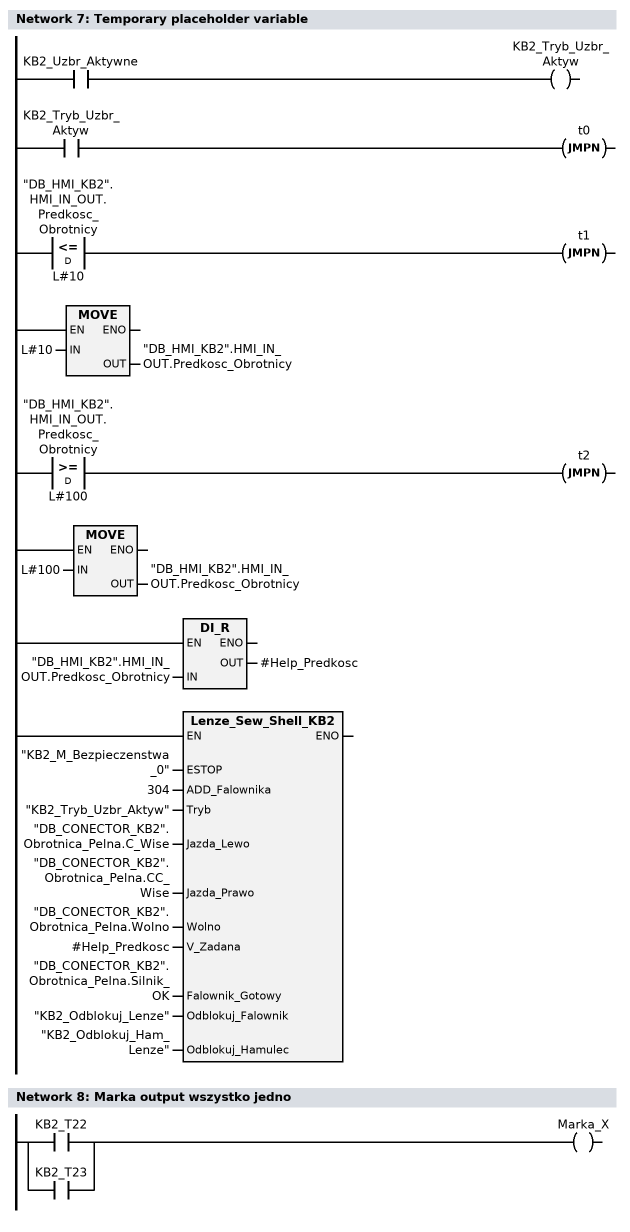
[picture p273: Przypis_Wyjsc_KB2 networks 7-8]
NETWORK
TITLE = Temporary placeholder variable
//Obrotnica Adres  9(Wirtualny)
// Dopasownie predkosci niskiej i wysokiej
      A     "KB2_Uzbr_Aktywne";
      =     "KB2_Tryb_Uzbr_Aktyw";
//************Przypisanie predkosci z panela*************
      A     "KB2_Tryb_Uzbr_Aktyw";
      JCN   t0;
//***Sprawdzenie czy predkosc nie jest za mala
      L     "DB_HMI_KB2".HMI_IN_OUT.Predkosc_Obrotnicy;
      L     L#10;
      <=D;
      JCN   t1;
      L     L#10;
      T     "DB_HMI_KB2".HMI_IN_OUT.Predkosc_Obrotnicy;
t1:   NOP   0;
//***Sprawdzenie czy predkosc nie jest za duza
      L     "DB_HMI_KB2".HMI_IN_OUT.Predkosc_Obrotnicy;
      L     L#100;
      >=D;
      JCN   t2;
      L     L#100;
      T     "DB_HMI_KB2".HMI_IN_OUT.Predkosc_Obrotnicy;
t2:   NOP   0;
//****Zamiana na real
t0:   NOP   0;
      L     "DB_HMI_KB2".HMI_IN_OUT.Predkosc_Obrotnicy;
      DTR;
      T     #Help_Predkosc;
//***Obsluga obrotnicy
      CALL  "Lenze_Sew_Shell_KB2" (
           ESTOP                    := "KB2_M_Bezpieczenstwa_0",
           ADD_Falownika            := 304,
           Tryb                     := "KB2_Tryb_Uzbr_Aktyw",
           Jazda_Lewo               := "DB_CONECTOR_KB2".Obrotnica_Pelna.C_Wise,
           Jazda_Prawo              := "DB_CONECTOR_KB2".Obrotnica_Pelna.CC_Wise,
           Wolno                    := "DB_CONECTOR_KB2".Obrotnica_Pelna.Wolno,
           V_Zadana                 := #Help_Predkosc,
           Falownik_Gotowy          := "DB_CONECTOR_KB2".Obrotnica_Pelna.Silnik_OK,
           Odblokuj_Falownik        := "KB2_Odblokuj_Lenze",
           Odblokuj_Hamulec         := "KB2_Odblokuj_Ham_Lenze");
NETWORK
TITLE = Marka output wszystko jedno
//Wpisz Timmer do rejestru
      O     "KB2_T22";
      O     "KB2_T23";
      =     "Marka_X";
END_FUNCTION

FUNCTION "Przypis_Wejsc_Buffory" : VOID	// FC 26
//Pobranie z bloku db stanu wejsc sieci asi i przyporzadkowanie do odpowiedniego 
//urzadzenia lini.
//
//
AUTHOR : Kng
NAME : Buff
VERSION : 0.1
VAR_TEMP
  Help_Bit_1 : BOOL ;
  Help_Bit_2 : BOOL ;
  Help_Word_1 : INT ;
  Help_Word_2 : INT ;
END_VAR
BEGIN
NETWORK
TITLE =
//Ten network celowo jest wolny
NETWORK
TITLE = Silnik ok
//Banda Adres 1 (Wirtualna) bo nalezy do segberta
NETWORK
TITLE = Silnik ok
//Banda Adres 2 
      A     "DB_ASi_Prosty_Odczyt_Buf".Adres_2_bit_0;
      =     "DB_CONNECTOR_BUFF".Banda_2.Silnik_OK;
      A     "DB_ASi_Prosty_Odczyt_Buf".Adres_2_bit_1;
      =     "DB_CONNECTOR_BUFF".Banda_2.Rezerwa_Silnik;
      A     "DB_ASi_Prosty_Odczyt_Buf".Adres_2_bit_2;
      =     "DB_CONNECTOR_BUFF".Banda_2.Foto_2;
      A     "DB_ASi_Prosty_Odczyt_Buf".Adres_2_bit_3;
      =     "DB_CONNECTOR_BUFF".Banda_2.Foto_1;
NETWORK
TITLE = Silnik ok
//Banda Adres 3
      A     "DB_ASi_Prosty_Odczyt_Buf".Adres_3_bit_0;
      =     "DB_CONNECTOR_BUFF".Banda_3.Silnik_OK;
      A     "DB_ASi_Prosty_Odczyt_Buf".Adres_3_bit_1;
      =     "DB_CONNECTOR_BUFF".Banda_3.Rezerwa_Silnik;
      A     "DB_ASi_Prosty_Odczyt_Buf".Adres_3_bit_2;
      =     "DB_CONNECTOR_BUFF".Banda_3.Foto_2;
      A     "DB_ASi_Prosty_Odczyt_Buf".Adres_3_bit_3;
      =     "DB_CONNECTOR_BUFF".Banda_3.Foto_1;
NETWORK
TITLE = Silnik ok
//Banda Adres 4 
      A     "DB_ASi_Prosty_Odczyt_Buf".Adres_4_bit_0;
      =     "DB_CONNECTOR_BUFF".Banda_4.Silnik_OK;
      A     "DB_ASi_Prosty_Odczyt_Buf".Adres_4_bit_1;
      =     "DB_CONNECTOR_BUFF".Banda_4.Rezerwa_Silnik;
      A     "DB_ASi_Prosty_Odczyt_Buf".Adres_4_bit_2;
      =     "DB_CONNECTOR_BUFF".Banda_4.Foto_2;
      A     "DB_ASi_Prosty_Odczyt_Buf".Adres_4_bit_3;
      =     "DB_CONNECTOR_BUFF".Banda_4.Foto_1;
NETWORK
TITLE = Silnik ok
//Banda Adres 5
      A     "DB_ASi_Prosty_Odczyt_Buf".Adres_5_bit_0;
      =     "DB_CONNECTOR_BUFF".Banda_5.Silnik_OK;
      A     "DB_ASi_Prosty_Odczyt_Buf".Adres_5_bit_1;
      =     "DB_CONNECTOR_BUFF".Banda_5.Rezerwa_Silnik;
      A     "DB_ASi_Prosty_Odczyt_Buf".Adres_5_bit_2;
      =     "DB_CONNECTOR_BUFF".Banda_5.Foto_2;
      A     "DB_ASi_Prosty_Odczyt_Buf".Adres_5_bit_3;
      =     "DB_CONNECTOR_BUFF".Banda_5.Foto_1;
NETWORK
TITLE = Silnik ok
//Banda Adres 6
      A     "DB_ASi_Prosty_Odczyt_Buf".Adres_6_bit_0;
      =     "DB_CONNECTOR_BUFF".Banda_6.Silnik_OK;
      A     "DB_ASi_Prosty_Odczyt_Buf".Adres_6_bit_1;
      =     "DB_CONNECTOR_BUFF".Banda_6.Rezerwa_Silnik;
      A     "DB_ASi_Prosty_Odczyt_Buf".Adres_6_bit_2;
      =     "DB_CONNECTOR_BUFF".Banda_6.Foto_2;
      A     "DB_ASi_Prosty_Odczyt_Buf".Adres_6_bit_3;
      =     "DB_CONNECTOR_BUFF".Banda_6.Foto_1;
NETWORK
TITLE = Silnik ok
//Banda   (shuttle)
NETWORK
TITLE = Silnik ok
//Banda adres 12
      A     "DB_ASi_Prosty_Odczyt_Buf".Adres_12_bit_0;
      =     "DB_CONNECTOR_BUFF".Banda_12.Silnik_OK;
      A     "DB_ASi_Prosty_Odczyt_Buf".Adres_12_bit_1;
      =     "DB_CONNECTOR_BUFF".Banda_12.Rezerwa_Silnik;
      A     "DB_ASi_Prosty_Odczyt_Buf".Adres_12_bit_2;
      =     "DB_CONNECTOR_BUFF".Banda_12.Foto_1;
      A     "DB_ASi_Prosty_Odczyt_Buf".Adres_12_bit_3;
      =     "DB_CONNECTOR_BUFF".Banda_12.Foto_2;
NETWORK
TITLE = Silnik ok
//Banda adres 13
      A     "DB_ASi_Prosty_Odczyt_Buf".Adres_13_bit_0;
      =     "DB_CONNECTOR_BUFF".banda_13.Silnik_OK;
      A     "DB_ASi_Prosty_Odczyt_Buf".Adres_13_bit_1;
      =     "DB_CONNECTOR_BUFF".banda_13.Rezerwa_Silnik;
      A     "DB_ASi_Prosty_Odczyt_Buf".Adres_13_bit_2;
      =     "DB_CONNECTOR_BUFF".banda_13.Foto_1;
      A     "DB_ASi_Prosty_Odczyt_Buf".Adres_13_bit_3;
      =     "DB_CONNECTOR_BUFF".banda_13.Foto_2;
NETWORK
TITLE = Silnik ok
//Banda 14
      A     "DB_ASi_Prosty_Odczyt_Buf".Adres_14_bit_0;
      =     "DB_CONNECTOR_BUFF".Banda_14.Silnik_OK;
      A     "DB_ASi_Prosty_Odczyt_Buf".Adres_14_bit_1;
      =     "DB_CONNECTOR_BUFF".Banda_14.Rezerwa_Silnik;
      A     "DB_ASi_Prosty_Odczyt_Buf".Adres_14_bit_2;
      =     "DB_CONNECTOR_BUFF".Banda_14.Foto_1;
      A     "DB_ASi_Prosty_Odczyt_Buf".Adres_14_bit_3;
      =     "DB_CONNECTOR_BUFF".Banda_14.Foto_2;
NETWORK
TITLE = Silnik ok
//Banda 15
      A     "DB_ASi_Prosty_Odczyt_Buf".Adres_15_bit_0;
      =     "DB_CONNECTOR_BUFF".Banda_15.Silnik_OK;
      A     "DB_ASi_Prosty_Odczyt_Buf".Adres_15_bit_1;
      =     "DB_CONNECTOR_BUFF".Banda_15.Rezerwa_Silnik;
      A     "DB_ASi_Prosty_Odczyt_Buf".Adres_15_bit_2;
      =     "DB_CONNECTOR_BUFF".Banda_15.Foto_1;
      A     "DB_ASi_Prosty_Odczyt_Buf".Adres_15_bit_3;
      =     "DB_CONNECTOR_BUFF".Banda_15.Foto_2;
NETWORK
TITLE = Silnik ok
//Banda 16
      A     "DB_ASi_Prosty_Odczyt_Buf".Adres_16_bit_0;
      =     "DB_CONNECTOR_BUFF".Banda_16.Silnik_OK;
      A     "DB_ASi_Prosty_Odczyt_Buf".Adres_16_bit_1;
      =     "DB_CONNECTOR_BUFF".Banda_16.Rezerwa_Silnik;
      A     "DB_ASi_Prosty_Odczyt_Buf".Adres_16_bit_2;
      =     "DB_CONNECTOR_BUFF".Banda_16.Foto_1;
      A     "DB_ASi_Prosty_Odczyt_Buf".Adres_16_bit_3;
      =     "DB_CONNECTOR_BUFF".Banda_16.Foto_2;
NETWORK
TITLE = Silnik ok
//Banda 7
      A     "DB_ASi_Prosty_Odczyt_Buf".Adres_7_bit_0;
      =     "DB_CONNECTOR_BUFF".Banda_7.Silnik_OK;
      A     "DB_ASi_Prosty_Odczyt_Buf".Adres_7_bit_1;
      =     "DB_CONNECTOR_BUFF".Banda_7.Rezerwa_Silnik;
      A     "DB_ASi_Prosty_Odczyt_Buf".Adres_7_bit_2;
      =     "DB_CONNECTOR_BUFF".Banda_7.Foto_1;
      A     "DB_ASi_Prosty_Odczyt_Buf".Adres_7_bit_3;
      =     "DB_CONNECTOR_BUFF".Banda_7.Foto_2;
NETWORK
TITLE = Silnik ok
//Banda 8
      A     "DB_ASi_Prosty_Odczyt_Buf".Adres_8_bit_0;
      =     "DB_CONNECTOR_BUFF".Banda_8.Silnik_OK;
      A     "DB_ASi_Prosty_Odczyt_Buf".Adres_8_bit_1;
      =     "DB_CONNECTOR_BUFF".Banda_8.Rezerwa_Silnik;
      A     "DB_ASi_Prosty_Odczyt_Buf".Adres_8_bit_2;
      =     "DB_CONNECTOR_BUFF".Banda_8.Foto_1;
      A     "DB_ASi_Prosty_Odczyt_Buf".Adres_8_bit_3;
      =     "DB_CONNECTOR_BUFF".Banda_8.Foto_2;
NETWORK
TITLE = Silnik ok
//Banda 17
      A     "DB_ASi_Prosty_Odczyt_Buf".Adres_17_bit_0;
      =     "DB_CONNECTOR_BUFF".Banda_17.Silnik_OK;
      A     "DB_ASi_Prosty_Odczyt_Buf".Adres_17_bit_1;
      =     "DB_CONNECTOR_BUFF".Banda_17.Rezerwa_Silnik;
      A     "DB_ASi_Prosty_Odczyt_Buf".Adres_17_bit_2;
      =     "DB_CONNECTOR_BUFF".Banda_17.Foto_1;
      A     "DB_ASi_Prosty_Odczyt_Buf".Adres_17_bit_3;
      =     "DB_CONNECTOR_BUFF".Banda_17.Foto_2;
NETWORK
TITLE = Silnik ok
//Banda 18
      A     "DB_ASi_Prosty_Odczyt_Buf".Adres_18_bit_0;
      =     "DB_CONNECTOR_BUFF".Banda_18.Silnik_OK;
      A     "DB_ASi_Prosty_Odczyt_Buf".Adres_18_bit_1;
      =     "DB_CONNECTOR_BUFF".Banda_18.Rezerwa_Silnik;
      A     "DB_ASi_Prosty_Odczyt_Buf".Adres_18_bit_2;
      =     "DB_CONNECTOR_BUFF".Banda_18.Foto_1;
      A     "DB_ASi_Prosty_Odczyt_Buf".Adres_18_bit_3;
      =     "DB_CONNECTOR_BUFF".Banda_18.Foto_2;
NETWORK
TITLE =
//20-Adres Not-Aus Pulpit
      A     "DB_ASi_Prosty_Odczyt_Buf".Adres_20_bit_0;
      =     "DB_CONNECTOR_BUFF".Not_Aus_1.EStop_Tor_1_1;
      A     "DB_ASi_Prosty_Odczyt_Buf".Adres_20_bit_1;
      =     "DB_CONNECTOR_BUFF".Not_Aus_1.EStop_Tor_1_2;
      A     "DB_ASi_Prosty_Odczyt_Buf".Adres_20_bit_2;
      =     "DB_CONNECTOR_BUFF".Not_Aus_1.EStop_Tor_2_1;
      A     "DB_ASi_Prosty_Odczyt_Buf".Adres_20_bit_3;
      =     "DB_CONNECTOR_BUFF".Not_Aus_1.EStop_Tor_2_2;
NETWORK
TITLE =
//24-Adres Not-Aus Wozek
      A     "DB_ASi_Prosty_Odczyt_Buf".Adres_24_bit_0;
      =     "DB_CONNECTOR_BUFF".Not_Aus_2.EStop_Tor_1_1;
      A     "DB_ASi_Prosty_Odczyt_Buf".Adres_24_bit_1;
      =     "DB_CONNECTOR_BUFF".Not_Aus_2.EStop_Tor_1_2;
      A     "DB_ASi_Prosty_Odczyt_Buf".Adres_24_bit_2;
      =     "DB_CONNECTOR_BUFF".Not_Aus_2.EStop_Tor_2_1;
      A     "DB_ASi_Prosty_Odczyt_Buf".Adres_24_bit_3;
      =     "DB_CONNECTOR_BUFF".Not_Aus_2.EStop_Tor_2_2;
END_FUNCTION

FUNCTION "Przypis_Wyjsc_Buffory" : VOID	// FC 27
AUTHOR : Kng
NAME : Buff
VERSION : 0.1
VAR_TEMP
  Temp_Word_1 : INT ;
  Help_Bit_1 : BOOL ;
END_VAR
BEGIN
NETWORK
TITLE =
//Ten Network celowo jest wolny
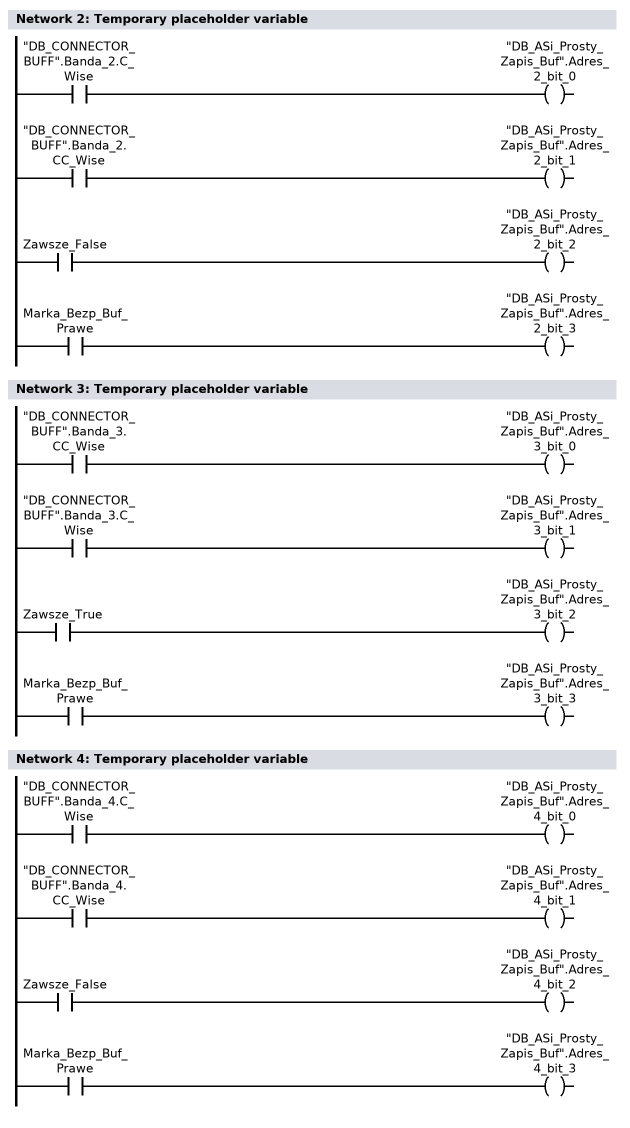
NETWORK
TITLE = Temporary placeholder variable
//Banda  Adres 2
//****************ClockWise*******************
      A     "DB_CONNECTOR_BUFF".Banda_2.C_Wise;	//C_Wise
      =     "DB_ASi_Prosty_Zapis_Buf".Adres_2_bit_0;
//****************CounterClockWise************
      A     "DB_CONNECTOR_BUFF".Banda_2.CC_Wise;
      =     "DB_ASi_Prosty_Zapis_Buf".Adres_2_bit_1;	//CC_Wise
//****************Wolno***********************
      A     "Zawsze_False";
      =     "DB_ASi_Prosty_Zapis_Buf".Adres_2_bit_2;	//Wolno
//****************Bit_Bezpieczenstwa**********
      A     "Marka_Bezp_Buf_Prawe";	//Safety
      =     "DB_ASi_Prosty_Zapis_Buf".Adres_2_bit_3;
NETWORK
TITLE = Temporary placeholder variable
//Banda Adres 3
//****************ClockWise*******************
      A     "DB_CONNECTOR_BUFF".Banda_3.CC_Wise;	//C_Wise
      =     "DB_ASi_Prosty_Zapis_Buf".Adres_3_bit_0;
//****************CounterClockWise************
      A     "DB_CONNECTOR_BUFF".Banda_3.C_Wise;
      =     "DB_ASi_Prosty_Zapis_Buf".Adres_3_bit_1;	//CC_Wise
//****************Wolno***********************
      A     "Zawsze_True";
      =     "DB_ASi_Prosty_Zapis_Buf".Adres_3_bit_2;	//Wolno
//****************Bit_Bezpieczenstwa**********
      A     "Marka_Bezp_Buf_Prawe";
      =     "DB_ASi_Prosty_Zapis_Buf".Adres_3_bit_3;
NETWORK
TITLE = Temporary placeholder variable
//Banda 4
//****************ClockWise*******************
      A     "DB_CONNECTOR_BUFF".Banda_4.C_Wise;	//C_Wise
      =     "DB_ASi_Prosty_Zapis_Buf".Adres_4_bit_0;
//****************CounterClockWise************
      A     "DB_CONNECTOR_BUFF".Banda_4.CC_Wise;
      =     "DB_ASi_Prosty_Zapis_Buf".Adres_4_bit_1;	//CC_Wise
//****************Wolno***********************
      A     "Zawsze_False";
      =     "DB_ASi_Prosty_Zapis_Buf".Adres_4_bit_2;	//Wolno
//****************Bit_Bezpieczenstwa**********
      A     "Marka_Bezp_Buf_Prawe";	//Safety
      =     "DB_ASi_Prosty_Zapis_Buf".Adres_4_bit_3;
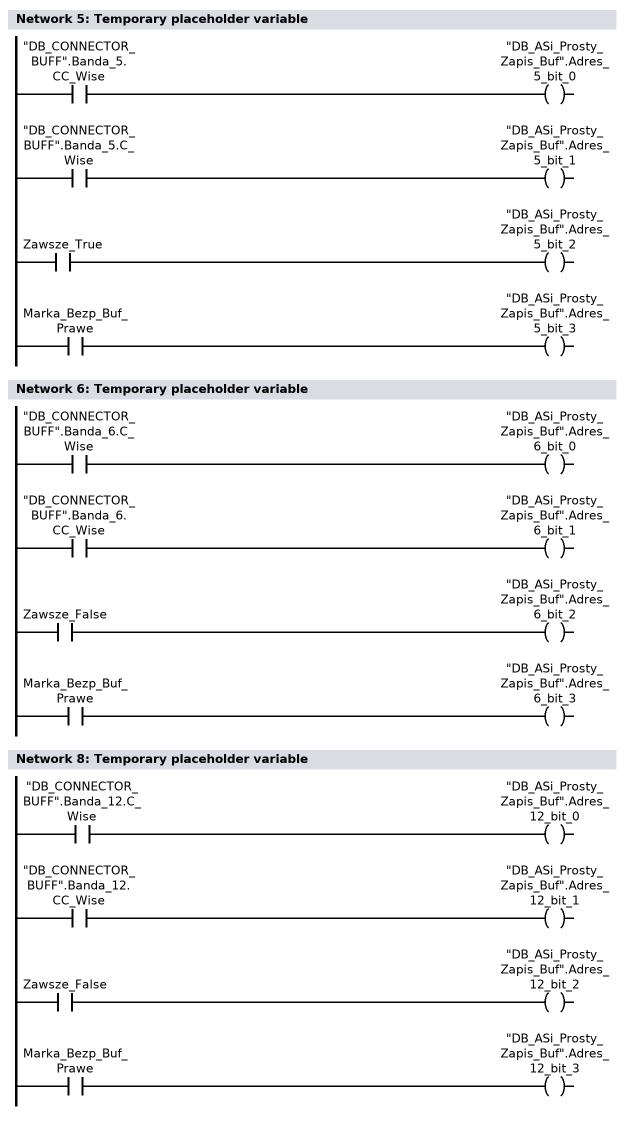
NETWORK
TITLE = Temporary placeholder variable
//Banda 5
//****************ClockWise*******************
      A     "DB_CONNECTOR_BUFF".Banda_5.CC_Wise;	//C_Wise
      =     "DB_ASi_Prosty_Zapis_Buf".Adres_5_bit_0;
//****************CounterClockWise************
      A     "DB_CONNECTOR_BUFF".Banda_5.C_Wise;
      =     "DB_ASi_Prosty_Zapis_Buf".Adres_5_bit_1;	//CC_Wise
//****************Wolno***********************
      A     "Zawsze_True";
      =     "DB_ASi_Prosty_Zapis_Buf".Adres_5_bit_2;	//Wolno
//****************Bit_Bezpieczenstwa**********
      A     "Marka_Bezp_Buf_Prawe";	//Safety
      =     "DB_ASi_Prosty_Zapis_Buf".Adres_5_bit_3;
NETWORK
TITLE = Temporary placeholder variable
//Banda 6
//****************ClockWise*******************
      A     "DB_CONNECTOR_BUFF".Banda_6.C_Wise;	//C_Wise
      =     "DB_ASi_Prosty_Zapis_Buf".Adres_6_bit_0;
//****************CounterClockWise************
      A     "DB_CONNECTOR_BUFF".Banda_6.CC_Wise;
      =     "DB_ASi_Prosty_Zapis_Buf".Adres_6_bit_1;	//CC_Wise
//****************Wolno***********************
      A     "Zawsze_False";
      =     "DB_ASi_Prosty_Zapis_Buf".Adres_6_bit_2;	//Wolno
//****************Bit_Bezpieczenstwa**********
      A     "Marka_Bezp_Buf_Prawe";	//Safety
      =     "DB_ASi_Prosty_Zapis_Buf".Adres_6_bit_3;
NETWORK
TITLE = Temporary placeholder variable
//Shuttle adres  
NETWORK
TITLE = Temporary placeholder variable
//Banda 12
//****************ClockWise*******************
      A     "DB_CONNECTOR_BUFF".Banda_12.C_Wise;	//C_Wise
      =     "DB_ASi_Prosty_Zapis_Buf".Adres_12_bit_0;
//****************CounterClockWise************
      A     "DB_CONNECTOR_BUFF".Banda_12.CC_Wise;
      =     "DB_ASi_Prosty_Zapis_Buf".Adres_12_bit_1;	//CC_Wise
//****************Wolno***********************
      A     "Zawsze_False";
      =     "DB_ASi_Prosty_Zapis_Buf".Adres_12_bit_2;	//Wolno
//****************Bit_Bezpieczenstwa**********
      A     "Marka_Bezp_Buf_Prawe";	//Safety
      =     "DB_ASi_Prosty_Zapis_Buf".Adres_12_bit_3;
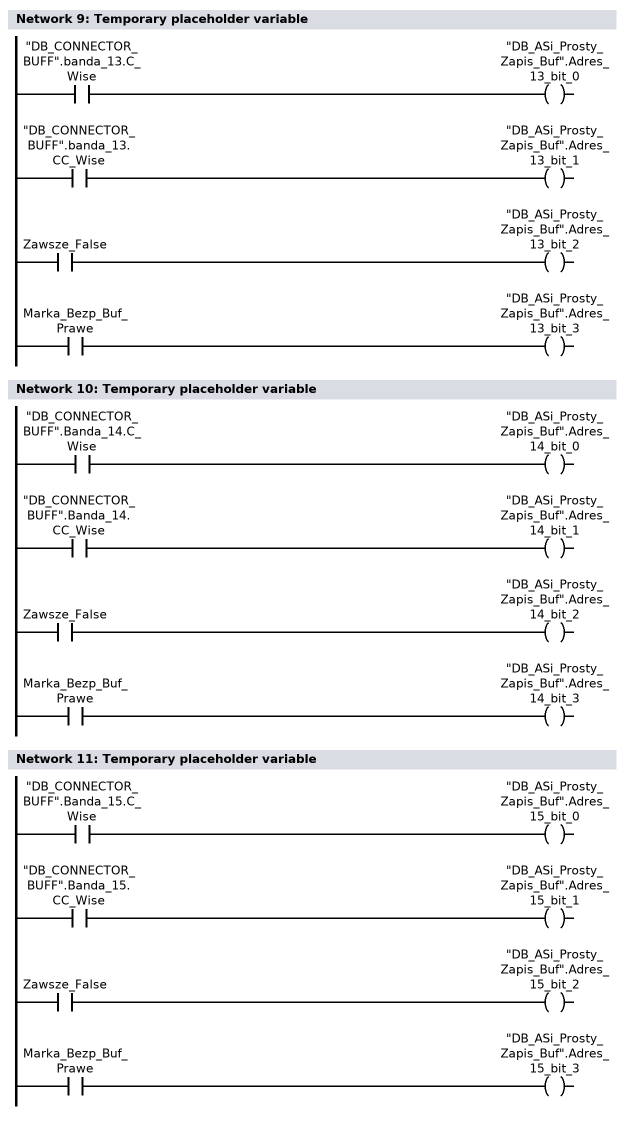
NETWORK
TITLE = Temporary placeholder variable
//Banda 13
//****************ClockWise*******************
      A     "DB_CONNECTOR_BUFF".banda_13.C_Wise;	//C_Wise
      =     "DB_ASi_Prosty_Zapis_Buf".Adres_13_bit_0;
//****************CounterClockWise************
      A     "DB_CONNECTOR_BUFF".banda_13.CC_Wise;
      =     "DB_ASi_Prosty_Zapis_Buf".Adres_13_bit_1;	//CC_Wise
//****************Wolno***********************
      A     "Zawsze_False";
      =     "DB_ASi_Prosty_Zapis_Buf".Adres_13_bit_2;	//Wolno
//****************Bit_Bezpieczenstwa**********
      A     "Marka_Bezp_Buf_Prawe";	//Safety
      =     "DB_ASi_Prosty_Zapis_Buf".Adres_13_bit_3;
NETWORK
TITLE = Temporary placeholder variable
//Banda 14
//****************ClockWise*******************
      A     "DB_CONNECTOR_BUFF".Banda_14.C_Wise;	//C_Wise
      =     "DB_ASi_Prosty_Zapis_Buf".Adres_14_bit_0;
//****************CounterClockWise************
      A     "DB_CONNECTOR_BUFF".Banda_14.CC_Wise;
      =     "DB_ASi_Prosty_Zapis_Buf".Adres_14_bit_1;	//CC_Wise
//****************Wolno***********************
      A     "Zawsze_False";
      =     "DB_ASi_Prosty_Zapis_Buf".Adres_14_bit_2;	//Wolno
//****************Bit_Bezpieczenstwa**********
      A     "Marka_Bezp_Buf_Prawe";	//Safety
      =     "DB_ASi_Prosty_Zapis_Buf".Adres_14_bit_3;
NETWORK
TITLE = Temporary placeholder variable
//Banda 15
//****************ClockWise*******************
      A     "DB_CONNECTOR_BUFF".Banda_15.C_Wise;	//C_Wise
      =     "DB_ASi_Prosty_Zapis_Buf".Adres_15_bit_0;
//****************CounterClockWise************
      A     "DB_CONNECTOR_BUFF".Banda_15.CC_Wise;
      =     "DB_ASi_Prosty_Zapis_Buf".Adres_15_bit_1;	//CC_Wise
//****************Wolno***********************
      A     "Zawsze_False";
      =     "DB_ASi_Prosty_Zapis_Buf".Adres_15_bit_2;	//Wolno
//****************Bit_Bezpieczenstwa**********
      A     "Marka_Bezp_Buf_Prawe";	//Safety
      =     "DB_ASi_Prosty_Zapis_Buf".Adres_15_bit_3;
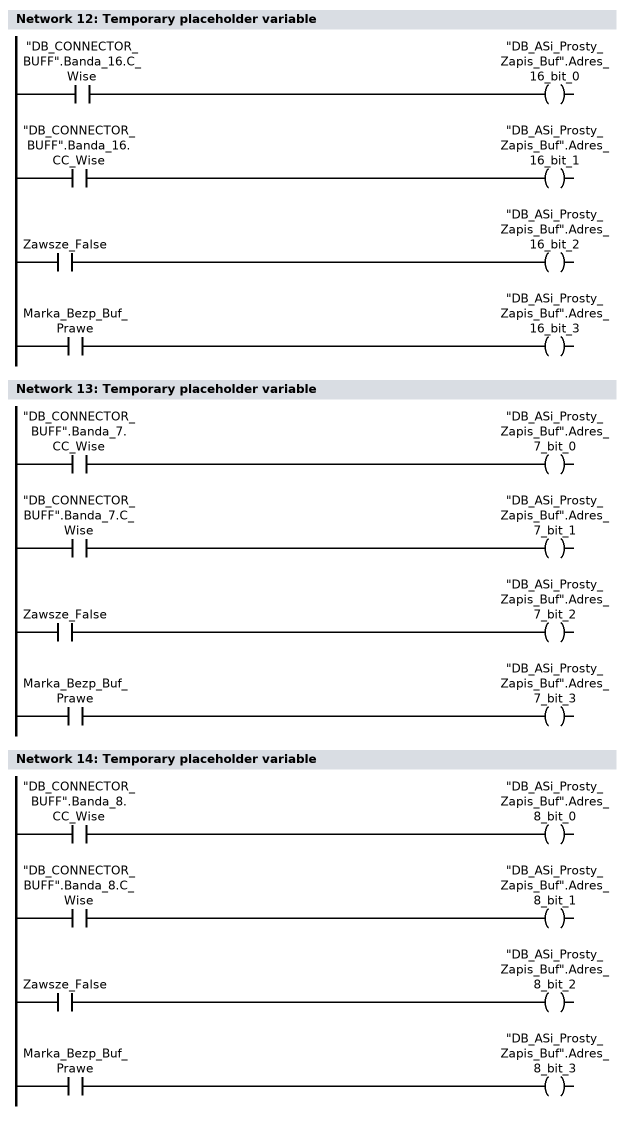
NETWORK
TITLE = Temporary placeholder variable
//Banda 16
//****************ClockWise*******************
      A     "DB_CONNECTOR_BUFF".Banda_16.C_Wise;	//C_Wise
      =     "DB_ASi_Prosty_Zapis_Buf".Adres_16_bit_0;
//****************CounterClockWise************
      A     "DB_CONNECTOR_BUFF".Banda_16.CC_Wise;
      =     "DB_ASi_Prosty_Zapis_Buf".Adres_16_bit_1;	//CC_Wise
//****************Wolno***********************
      A     "Zawsze_False";
      =     "DB_ASi_Prosty_Zapis_Buf".Adres_16_bit_2;	//Wolno
//****************Bit_Bezpieczenstwa**********
      A     "Marka_Bezp_Buf_Prawe";	//Safety
      =     "DB_ASi_Prosty_Zapis_Buf".Adres_16_bit_3;
NETWORK
TITLE = Temporary placeholder variable
//Banda 7
//****************ClockWise*******************
      A     "DB_CONNECTOR_BUFF".Banda_7.CC_Wise;	//C_Wise
      =     "DB_ASi_Prosty_Zapis_Buf".Adres_7_bit_0;
//****************CounterClockWise************
      A     "DB_CONNECTOR_BUFF".Banda_7.C_Wise;
      =     "DB_ASi_Prosty_Zapis_Buf".Adres_7_bit_1;	//CC_Wise
//****************Wolno***********************
      A     "Zawsze_False";
      =     "DB_ASi_Prosty_Zapis_Buf".Adres_7_bit_2;	//Wolno
//****************Bit_Bezpieczenstwa**********
      A     "Marka_Bezp_Buf_Prawe";	//Safety
      =     "DB_ASi_Prosty_Zapis_Buf".Adres_7_bit_3;
NETWORK
TITLE = Temporary placeholder variable
//Banda 8
//****************ClockWise*******************
      A     "DB_CONNECTOR_BUFF".Banda_8.CC_Wise;	//C_Wise
      =     "DB_ASi_Prosty_Zapis_Buf".Adres_8_bit_0;
//****************CounterClockWise************
      A     "DB_CONNECTOR_BUFF".Banda_8.C_Wise;
      =     "DB_ASi_Prosty_Zapis_Buf".Adres_8_bit_1;	//CC_Wise
//****************Wolno***********************
      A     "Zawsze_False";
      =     "DB_ASi_Prosty_Zapis_Buf".Adres_8_bit_2;	//Wolno
//****************Bit_Bezpieczenstwa**********
      A     "Marka_Bezp_Buf_Prawe";	//Safety
      =     "DB_ASi_Prosty_Zapis_Buf".Adres_8_bit_3;
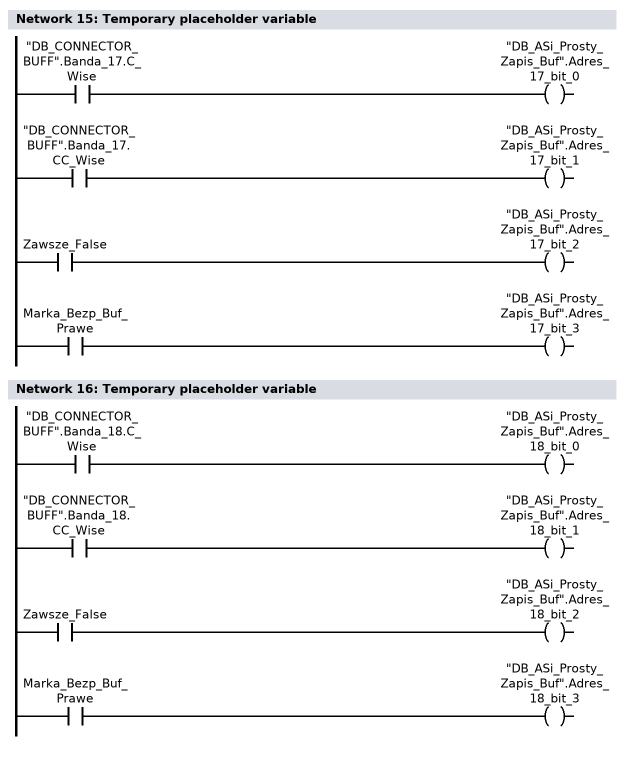
NETWORK
TITLE = Temporary placeholder variable
//Banda 17
//****************ClockWise*******************
      A     "DB_CONNECTOR_BUFF".Banda_17.C_Wise;	//C_Wise
      =     "DB_ASi_Prosty_Zapis_Buf".Adres_17_bit_0;
//****************CounterClockWise************
      A     "DB_CONNECTOR_BUFF".Banda_17.CC_Wise;
      =     "DB_ASi_Prosty_Zapis_Buf".Adres_17_bit_1;	//CC_Wise
//****************Wolno***********************
      A     "Zawsze_False";
      =     "DB_ASi_Prosty_Zapis_Buf".Adres_17_bit_2;	//Wolno
//****************Bit_Bezpieczenstwa**********
      A     "Marka_Bezp_Buf_Prawe";	//Safety
      =     "DB_ASi_Prosty_Zapis_Buf".Adres_17_bit_3;
NETWORK
TITLE = Temporary placeholder variable
//Banda 18
//****************ClockWise*******************
      A     "DB_CONNECTOR_BUFF".Banda_18.C_Wise;	//C_Wise
      =     "DB_ASi_Prosty_Zapis_Buf".Adres_18_bit_0;
//****************CounterClockWise************
      A     "DB_CONNECTOR_BUFF".Banda_18.CC_Wise;
      =     "DB_ASi_Prosty_Zapis_Buf".Adres_18_bit_1;	//CC_Wise
//****************Wolno***********************
      A     "Zawsze_False";
      =     "DB_ASi_Prosty_Zapis_Buf".Adres_18_bit_2;	//Wolno
//****************Bit_Bezpieczenstwa**********
      A     "Marka_Bezp_Buf_Prawe";	//Safety
      =     "DB_ASi_Prosty_Zapis_Buf".Adres_18_bit_3;
NETWORK
TITLE =
END_FUNCTION

FUNCTION "Ruch_Palety" : VOID	// FC 40
VERSION : 0.1
VAR_INPUT
  Foto_Wlotu : BOOL ;
  Foto_Wylotu : BOOL ;
  Foto_Wlotu_Nast_Palety : BOOL ;
  HMI_uzbrajanie : BOOL ;
  HMI_foliowanie : BOOL ;
  HMI_deklowanie : BOOL ;
  HMI_wiaz_wzdl : BOOL ;
  HMI_wiaz_poprz : BOOL ;
END_VAR
VAR_OUTPUT
  Znacznik_Ruchu : BYTE ;
  Status_Uzbrajania : BOOL ;
  Status_Foliowania : BOOL ;
  Status_Deklowania : BOOL ;
  Status_Wiaz_wzdl : BOOL ;
  Status_Wiaz_poprz : BOOL ;
  Status_Widocznosci : BOOL ;
END_VAR
VAR_TEMP
  case_1 : BOOL ;
  case_2 : BOOL ;
  case_3 : BOOL ;
END_VAR
BEGIN
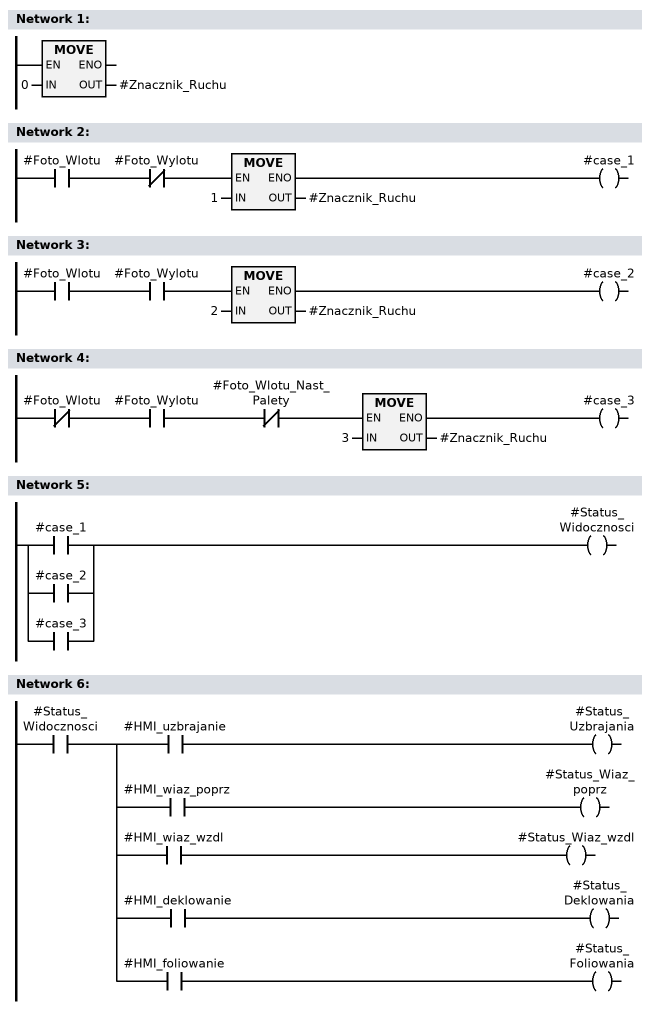
NETWORK
TITLE =
      L     0;
      T     #Znacznik_Ruchu;
      NOP   0;
NETWORK
TITLE =
      A     #Foto_Wlotu;
      AN    #Foto_Wylotu;
      JNB   _001;
      L     1;
      T     #Znacznik_Ruchu;
      SET;
      SAVE;
      CLR;
_001: A     BR;
      =     #case_1;
NETWORK
TITLE =
      A     #Foto_Wlotu;
      A     #Foto_Wylotu;
      JNB   _002;
      L     2;
      T     #Znacznik_Ruchu;
      SET;
      SAVE;
      CLR;
_002: A     BR;
      =     #case_2;
NETWORK
TITLE =
      AN    #Foto_Wlotu;
      A     #Foto_Wylotu;
      AN    #Foto_Wlotu_Nast_Palety;
      JNB   _003;
      L     3;
      T     #Znacznik_Ruchu;
      SET;
      SAVE;
      CLR;
_003: A     BR;
      =     #case_3;
NETWORK
TITLE =
      O     #case_1;
      O     #case_2;
      O     #case_3;
      =     #Status_Widocznosci;
NETWORK
TITLE =
      A     #Status_Widocznosci;
      =     L 1.0;
      A     L 1.0;
      A     #HMI_uzbrajanie;
      =     #Status_Uzbrajania;
      A     L 1.0;
      A     #HMI_wiaz_poprz;
      =     #Status_Wiaz_poprz;
      A     L 1.0;
      A     #HMI_wiaz_wzdl;
      =     #Status_Wiaz_wzdl;
      A     L 1.0;
      A     #HMI_deklowanie;
      =     #Status_Deklowania;
      A     L 1.0;
      A     #HMI_foliowanie;
      =     #Status_Foliowania;
END_FUNCTION

FUNCTION "Ruch_Palety_Winda" : VOID	// FC 41
VERSION : 0.1
VAR_INPUT
  Foto_Wlotu : BOOL ;
  Foto_Wylotu : BOOL ;
  Foto_Wlotu_Nast_Palety : BOOL ;
  HMI_uzbrajanie : BOOL ;
  HMI_foliowanie : BOOL ;
  HMI_deklowanie : BOOL ;
  HMI_wiaz_wzdl : BOOL ;
  HMI_wiaz_poprz : BOOL ;
END_VAR
VAR_OUTPUT
  Znacznik_Ruchu : INT ;
  Status_Uzbrajania : BOOL ;
  Status_Foliowania : BOOL ;
  Status_Deklowania : BOOL ;
  Status_Wiaz_wzdl : BOOL ;
  Status_Wiaz_poprz : BOOL ;
  Status_Widocznosci : BOOL ;
END_VAR
VAR_TEMP
  case_1 : BOOL ;
  case_2 : BOOL ;
  case_3 : BOOL ;
END_VAR
BEGIN
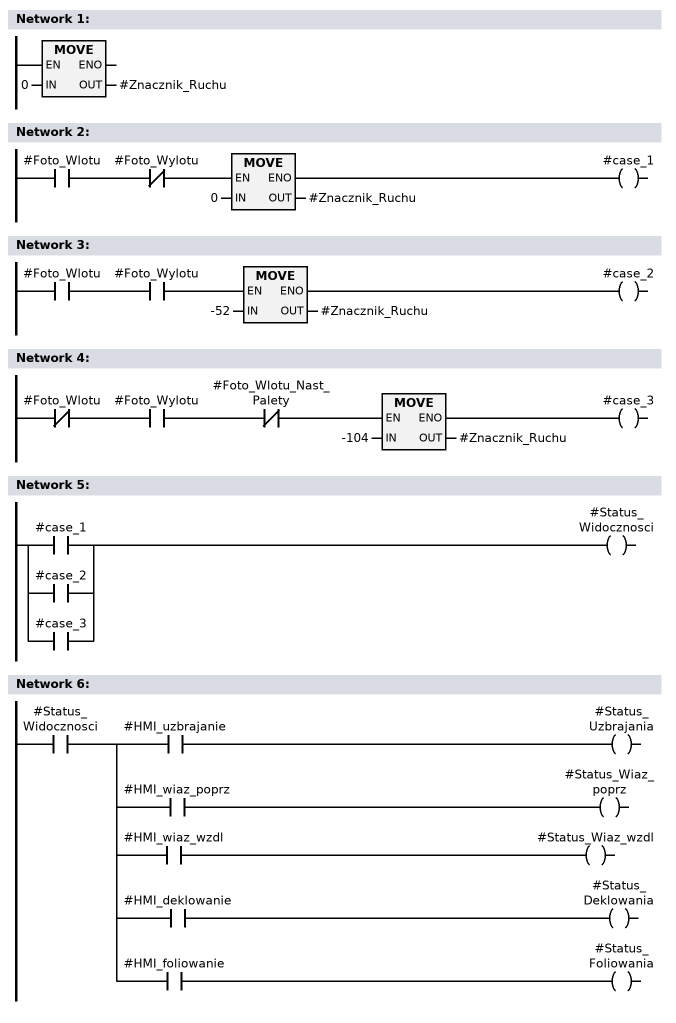
NETWORK
TITLE =
      L     0;
      T     #Znacznik_Ruchu;
      NOP   0;
NETWORK
TITLE =
      A     #Foto_Wlotu;
      AN    #Foto_Wylotu;
      JNB   _001;
      L     0;
      T     #Znacznik_Ruchu;
      SET;
      SAVE;
      CLR;
_001: A     BR;
      =     #case_1;
NETWORK
TITLE =
      A     #Foto_Wlotu;
      A     #Foto_Wylotu;
      JNB   _002;
      L     -52;
      T     #Znacznik_Ruchu;
      SET;
      SAVE;
      CLR;
_002: A     BR;
      =     #case_2;
NETWORK
TITLE =
      AN    #Foto_Wlotu;
      A     #Foto_Wylotu;
      AN    #Foto_Wlotu_Nast_Palety;
      JNB   _003;
      L     -104;
      T     #Znacznik_Ruchu;
      SET;
      SAVE;
      CLR;
_003: A     BR;
      =     #case_3;
NETWORK
TITLE =
      O     #case_1;
      O     #case_2;
      O     #case_3;
      =     #Status_Widocznosci;
NETWORK
TITLE =
      A     #Status_Widocznosci;
      =     L 1.0;
      A     L 1.0;
      A     #HMI_uzbrajanie;
      =     #Status_Uzbrajania;
      A     L 1.0;
      A     #HMI_wiaz_poprz;
      =     #Status_Wiaz_poprz;
      A     L 1.0;
      A     #HMI_wiaz_wzdl;
      =     #Status_Wiaz_wzdl;
      A     L 1.0;
      A     #HMI_deklowanie;
      =     #Status_Deklowania;
      A     L 1.0;
      A     #HMI_foliowanie;
      =     #Status_Foliowania;
END_FUNCTION

FUNCTION "ASI_Prosty_Odczyt" : VOID	// FC 82
//Pobieranie danych z modulu ASI CP 342-2
AUTHOR : Kng
FAMILY : Asi_fun
NAME : r_ASi
VERSION : 0.1
VAR_INPUT
  CP_Adr : INT ;
  DB_Nr : BLOCK_DB ;
END_VAR
BEGIN
NETWORK
TITLE =
      OPN   #DB_Nr;	// Nr bloku db
      L     #CP_Adr;	// Adres urzadzenia
      SLD   3;	//Przejscie na wskaznik
      LAR1;
      L     0;
      LAR2;
//Przepisanie z modulu Asi do bloku danych
      L     PID [AR1,P#0.0];
      T     DBD [AR2,P#0.0];
      L     PID [AR1,P#4.0];
      T     DBD [AR2,P#4.0];
      L     PID [AR1,P#8.0];
      T     DBD [AR2,P#8.0];
      L     PID [AR1,P#12.0];
      T     DBD [AR2,P#12.0];
END_FUNCTION

FUNCTION "ASI_Prosty_Zapis" : VOID	// FC 83
//Pobieranie danych z modulu ASI CP 342-2
AUTHOR : Kng
FAMILY : Asi_fun
NAME : w_ASi
VERSION : 0.1
VAR_INPUT
  CP_Adr : INT ;
  DB_Nr : BLOCK_DB ;
END_VAR
BEGIN
NETWORK
TITLE =
      OPN   #DB_Nr;	// Nr bloku db
      L     #CP_Adr;	// Adres urzadzenia
      SLD   3;	//Przejscie na wskaznik
      LAR1;
      L     0;
      LAR2;
//Przepisanie wartosci z bloku danych do modulu ASI
      L     DBD [AR2,P#0.0];
      T     PQD [AR1,P#0.0];
      L     DBD [AR2,P#4.0];
      T     PQD [AR1,P#4.0];
      L     DBD [AR2,P#8.0];
      T     PQD [AR1,P#8.0];
      L     DBD [AR2,P#12.0];
      T     PQD [AR1,P#12.0];
END_FUNCTION

FUNCTION "Opoznienie_Wylotu" : VOID	// FC 85
VERSION : 0.1
VAR_INPUT
  Wejscie : BOOL ;	//Fotokomorka
  Timmer_1 : TIMER ;
  Timmer_2 : TIMER ;
END_VAR
VAR_OUTPUT
  Wyjscie : BOOL ;
END_VAR
VAR_IN_OUT
  Zmienna : BOOL ;
END_VAR
BEGIN
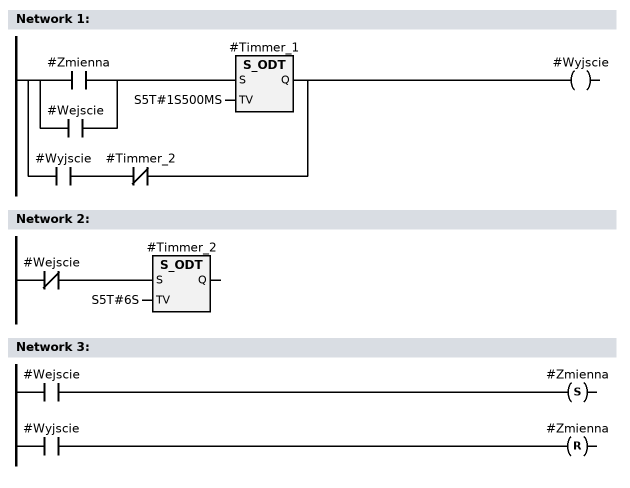
NETWORK
TITLE =
      O(;
      A(;
      O     #Zmienna;
      O     #Wejscie;
      );
      L     S5T#1S500MS;
      SD    #Timmer_1;
      NOP   0;
      NOP   0;
      NOP   0;
      A     #Timmer_1;
      );
      O;
      A     #Wyjscie;
      AN    #Timmer_2;
      =     #Wyjscie;
NETWORK
TITLE =
      AN    #Wejscie;
      L     S5T#6S;
      SD    #Timmer_2;
      NOP   0;
      NOP   0;
      NOP   0;
      NOP   0;
NETWORK
TITLE =
      A     #Wejscie;
      S     #Zmienna;
      A     #Wyjscie;
      R     #Zmienna;
      NOP   0;
END_FUNCTION

FUNCTION "FC_Bledy_KB1" : VOID	// FC 117
//Funkcja ta zawiera informacje o bledach na kb2
VERSION : 0.1
BEGIN
NETWORK
TITLE =
//Ten network celowo jest wolny
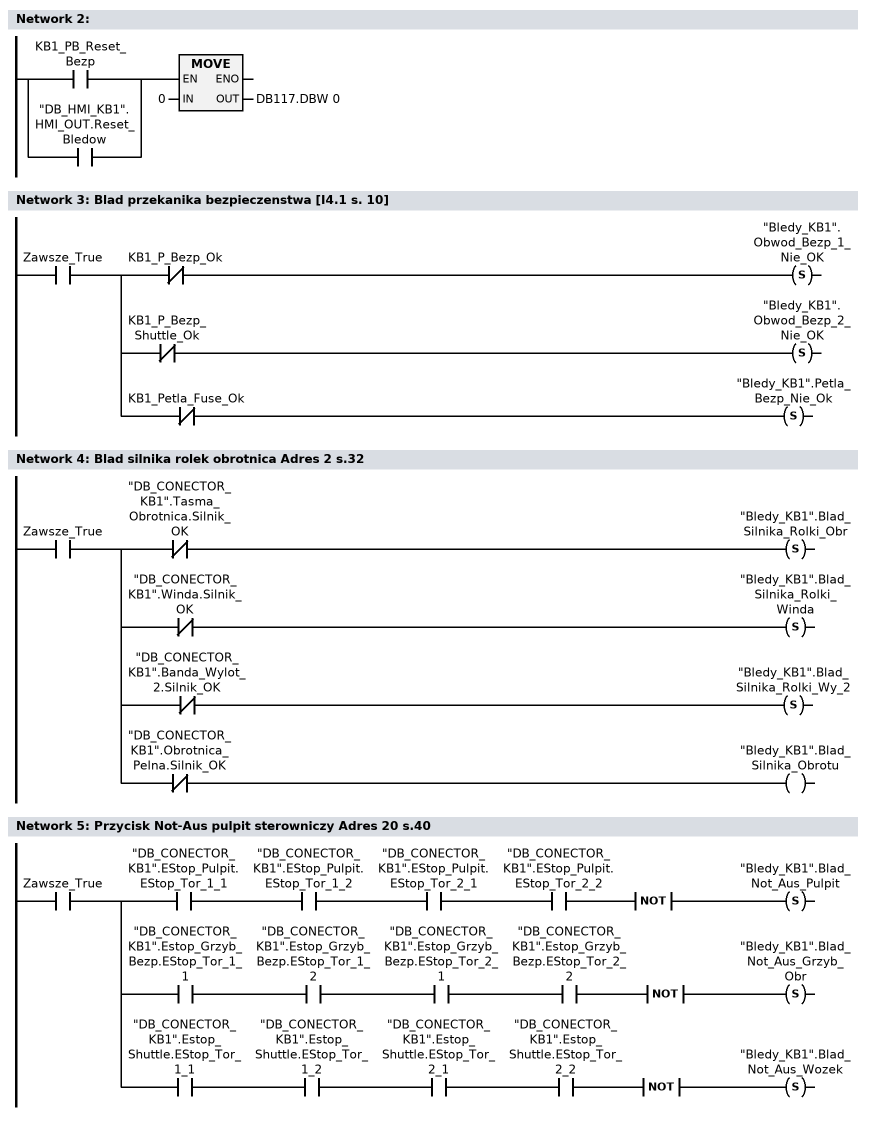
NETWORK
TITLE =
//Kasowanie bledow
      A(;
      O     "KB1_PB_Reset_Bezp";
      O     "DB_HMI_KB1".HMI_OUT.Reset_Bledow;
      );
      JNB   _001;
      L     0;
      T     DB117.DBW 0;
_001: NOP   0;
NETWORK
TITLE = Blad przekanika bezpieczenstwa [I4.1 s. 10]
      A     "Zawsze_True";
      =     L 0.0;
      A     L 0.0;
      AN    "KB1_P_Bezp_Ok";
      S     "Bledy_KB1".Obwod_Bezp_1_Nie_OK;
      A     L 0.0;
      AN    "KB1_P_Bezp_Shuttle_Ok";
      S     "Bledy_KB1".Obwod_Bezp_2_Nie_OK;
      A     L 0.0;
      AN    "KB1_Petla_Fuse_Ok";
      S     "Bledy_KB1".Petla_Bezp_Nie_Ok;
NETWORK
TITLE = Blad silnika rolek obrotnica Adres 2 s.32
//Bledy silnikow 
      A     "Zawsze_True";
      =     L 0.0;
      A     L 0.0;
      AN    "DB_CONECTOR_KB1".Tasma_Obrotnica.Silnik_OK;
      S     "Bledy_KB1".Blad_Silnika_Rolki_Obr;
      A     L 0.0;
      AN    "DB_CONECTOR_KB1".Winda.Silnik_OK;
      S     "Bledy_KB1".Blad_Silnika_Rolki_Winda;
      A     L 0.0;
      AN    "DB_CONECTOR_KB1".Banda_Wylot_2.Silnik_OK;
      S     "Bledy_KB1".Blad_Silnika_Rolki_Wy_2;
      A     L 0.0;
      AN    "DB_CONECTOR_KB1".Obrotnica_Pelna.Silnik_OK;
      =     "Bledy_KB1".Blad_Silnika_Obrotu;
NETWORK
TITLE = Przycisk Not-Aus pulpit sterowniczy Adres 20 s.40
//Bledy not aus
      A     "Zawsze_True";
      =     L 0.0;
      A     L 0.0;
      A     "DB_CONECTOR_KB1".EStop_Pulpit.EStop_Tor_1_1;
      A     "DB_CONECTOR_KB1".EStop_Pulpit.EStop_Tor_1_2;
      A     "DB_CONECTOR_KB1".EStop_Pulpit.EStop_Tor_2_1;
      A     "DB_CONECTOR_KB1".EStop_Pulpit.EStop_Tor_2_2;
      NOT;
      S     "Bledy_KB1".Blad_Not_Aus_Pulpit;
      A     L 0.0;
      A     "DB_CONECTOR_KB1".Estop_Grzyb_Bezp.EStop_Tor_1_1;
      A     "DB_CONECTOR_KB1".Estop_Grzyb_Bezp.EStop_Tor_1_2;
      A     "DB_CONECTOR_KB1".Estop_Grzyb_Bezp.EStop_Tor_2_1;
      A     "DB_CONECTOR_KB1".Estop_Grzyb_Bezp.EStop_Tor_2_2;
      NOT;
      S     "Bledy_KB1".Blad_Not_Aus_Grzyb_Obr;
      A     L 0.0;
      A     "DB_CONECTOR_KB1".Estop_Shuttle.EStop_Tor_1_1;
      A     "DB_CONECTOR_KB1".Estop_Shuttle.EStop_Tor_1_2;
      A     "DB_CONECTOR_KB1".Estop_Shuttle.EStop_Tor_2_1;
      A     "DB_CONECTOR_KB1".Estop_Shuttle.EStop_Tor_2_2;
      NOT;
      S     "Bledy_KB1".Blad_Not_Aus_Wozek;
END_FUNCTION

FUNCTION "FC_Bledy_KB2" : VOID	// FC 118
//Funkcja ta zawiera informacje o bledach na kb2
VERSION : 0.1
BEGIN
NETWORK
TITLE =
//Ten network celowo jest wolny
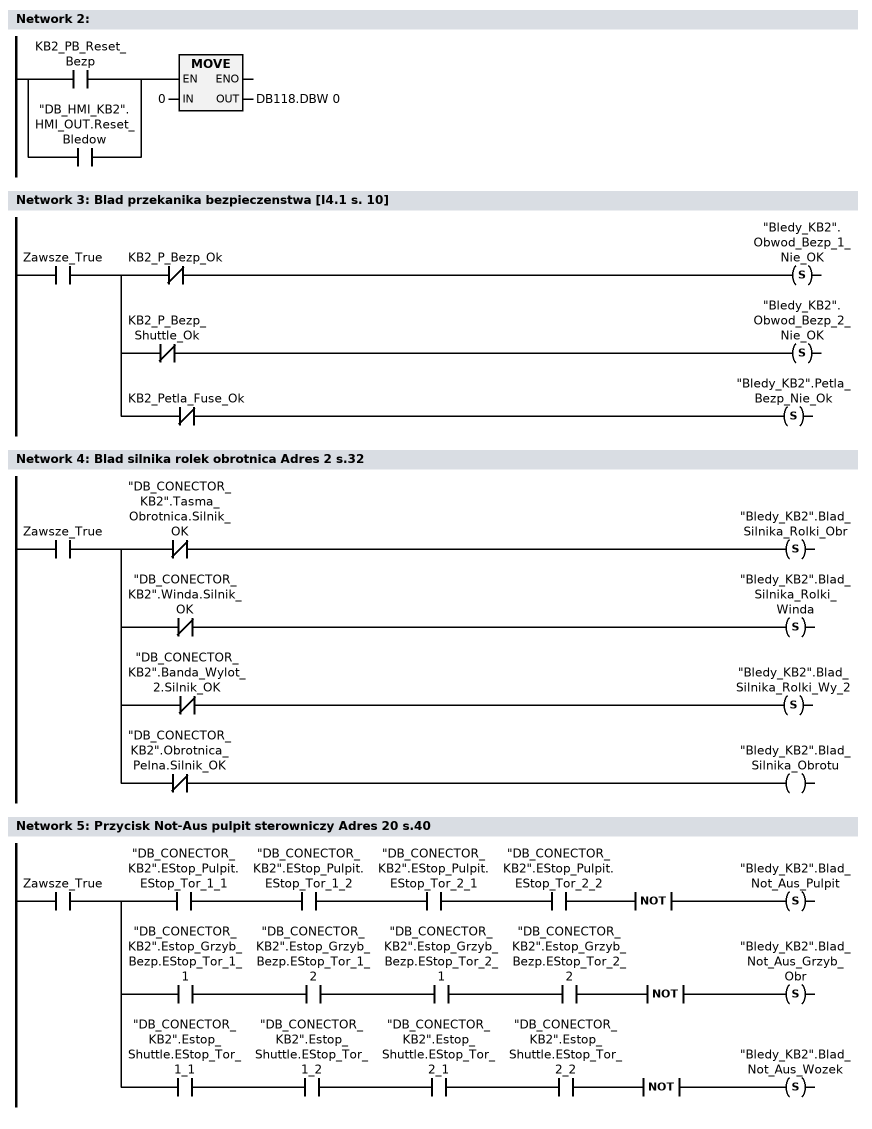
NETWORK
TITLE =
//Kasowanie bledow
      A(;
      O     "KB2_PB_Reset_Bezp";
      O     "DB_HMI_KB2".HMI_OUT.Reset_Bledow;
      );
      JNB   _001;
      L     0;
      T     DB118.DBW 0;
_001: NOP   0;
NETWORK
TITLE = Blad przekanika bezpieczenstwa [I4.1 s. 10]
      A     "Zawsze_True";
      =     L 0.0;
      A     L 0.0;
      AN    "KB2_P_Bezp_Ok";
      S     "Bledy_KB2".Obwod_Bezp_1_Nie_OK;
      A     L 0.0;
      AN    "KB2_P_Bezp_Shuttle_Ok";
      S     "Bledy_KB2".Obwod_Bezp_2_Nie_OK;
      A     L 0.0;
      AN    "KB2_Petla_Fuse_Ok";
      S     "Bledy_KB2".Petla_Bezp_Nie_Ok;
NETWORK
TITLE = Blad silnika rolek obrotnica Adres 2 s.32
//Bledy silnikow 
      A     "Zawsze_True";
      =     L 0.0;
      A     L 0.0;
      AN    "DB_CONECTOR_KB2".Tasma_Obrotnica.Silnik_OK;
      S     "Bledy_KB2".Blad_Silnika_Rolki_Obr;
      A     L 0.0;
      AN    "DB_CONECTOR_KB2".Winda.Silnik_OK;
      S     "Bledy_KB2".Blad_Silnika_Rolki_Winda;
      A     L 0.0;
      AN    "DB_CONECTOR_KB2".Banda_Wylot_2.Silnik_OK;
      S     "Bledy_KB2".Blad_Silnika_Rolki_Wy_2;
      A     L 0.0;
      AN    "DB_CONECTOR_KB2".Obrotnica_Pelna.Silnik_OK;
      =     "Bledy_KB2".Blad_Silnika_Obrotu;
NETWORK
TITLE = Przycisk Not-Aus pulpit sterowniczy Adres 20 s.40
//Bledy not aus
      A     "Zawsze_True";
      =     L 0.0;
      A     L 0.0;
      A     "DB_CONECTOR_KB2".EStop_Pulpit.EStop_Tor_1_1;
      A     "DB_CONECTOR_KB2".EStop_Pulpit.EStop_Tor_1_2;
      A     "DB_CONECTOR_KB2".EStop_Pulpit.EStop_Tor_2_1;
      A     "DB_CONECTOR_KB2".EStop_Pulpit.EStop_Tor_2_2;
      NOT;
      S     "Bledy_KB2".Blad_Not_Aus_Pulpit;
      A     L 0.0;
      A     "DB_CONECTOR_KB2".Estop_Grzyb_Bezp.EStop_Tor_1_1;
      A     "DB_CONECTOR_KB2".Estop_Grzyb_Bezp.EStop_Tor_1_2;
      A     "DB_CONECTOR_KB2".Estop_Grzyb_Bezp.EStop_Tor_2_1;
      A     "DB_CONECTOR_KB2".Estop_Grzyb_Bezp.EStop_Tor_2_2;
      NOT;
      S     "Bledy_KB2".Blad_Not_Aus_Grzyb_Obr;
      A     L 0.0;
      A     "DB_CONECTOR_KB2".Estop_Shuttle.EStop_Tor_1_1;
      A     "DB_CONECTOR_KB2".Estop_Shuttle.EStop_Tor_1_2;
      A     "DB_CONECTOR_KB2".Estop_Shuttle.EStop_Tor_2_1;
      A     "DB_CONECTOR_KB2".Estop_Shuttle.EStop_Tor_2_2;
      NOT;
      S     "Bledy_KB2".Blad_Not_Aus_Wozek;
END_FUNCTION

FUNCTION "FC_Bledy_Buff" : VOID	// FC 119
//Funkcja ta zawiera informacje o bledach na kb2
VERSION : 0.1
BEGIN
NETWORK
TITLE =
//Ten network celowo jest wolny
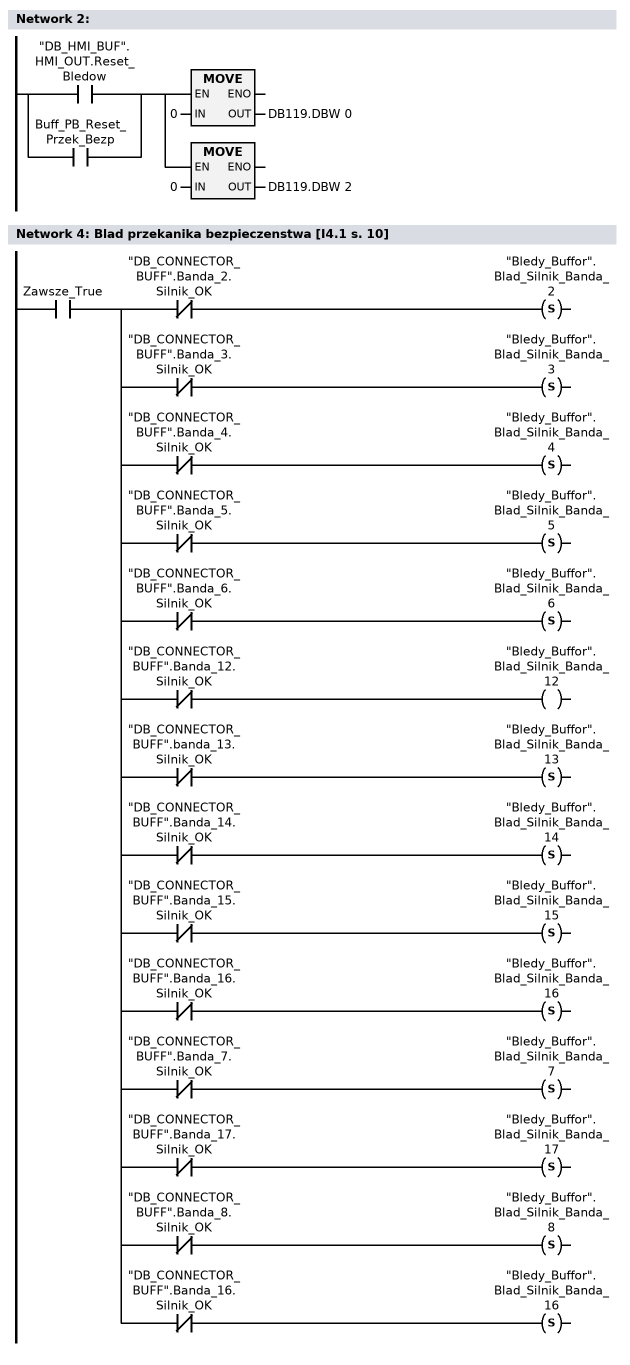
NETWORK
TITLE =
//Kasowanie bledow
      O     "DB_HMI_BUF".HMI_OUT.Reset_Bledow;
      O     "Buff_PB_Reset_Przek_Bezp";
      =     L 0.0;
      A     L 0.0;
      JNB   _001;
      L     0;
      T     DB119.DBW 0;
_001: NOP   0;
      A     L 0.0;
      JNB   _002;
      L     0;
      T     DB119.DBW 2;
_002: NOP   0;
NETWORK
TITLE =
NETWORK
TITLE = Blad przekanika bezpieczenstwa [I4.1 s. 10]
      A     "Zawsze_True";
      =     L 0.0;
      A     L 0.0;
      AN    "DB_CONNECTOR_BUFF".Banda_2.Silnik_OK;
      S     "Bledy_Buffor".Blad_Silnik_Banda_2;
      A     L 0.0;
      AN    "DB_CONNECTOR_BUFF".Banda_3.Silnik_OK;
      S     "Bledy_Buffor".Blad_Silnik_Banda_3;
      A     L 0.0;
      AN    "DB_CONNECTOR_BUFF".Banda_4.Silnik_OK;
      S     "Bledy_Buffor".Blad_Silnik_Banda_4;
      A     L 0.0;
      AN    "DB_CONNECTOR_BUFF".Banda_5.Silnik_OK;
      S     "Bledy_Buffor".Blad_Silnik_Banda_5;
      A     L 0.0;
      AN    "DB_CONNECTOR_BUFF".Banda_6.Silnik_OK;
      S     "Bledy_Buffor".Blad_Silnik_Banda_6;
      A     L 0.0;
      AN    "DB_CONNECTOR_BUFF".Banda_12.Silnik_OK;
      =     "Bledy_Buffor".Blad_Silnik_Banda_12;
      A     L 0.0;
      AN    "DB_CONNECTOR_BUFF".banda_13.Silnik_OK;
      S     "Bledy_Buffor".Blad_Silnik_Banda_13;
      A     L 0.0;
      AN    "DB_CONNECTOR_BUFF".Banda_14.Silnik_OK;
      S     "Bledy_Buffor".Blad_Silnik_Banda_14;
      A     L 0.0;
      AN    "DB_CONNECTOR_BUFF".Banda_15.Silnik_OK;
      S     "Bledy_Buffor".Blad_Silnik_Banda_15;
      A     L 0.0;
      AN    "DB_CONNECTOR_BUFF".Banda_16.Silnik_OK;
      S     "Bledy_Buffor".Blad_Silnik_Banda_16;
      A     L 0.0;
      AN    "DB_CONNECTOR_BUFF".Banda_7.Silnik_OK;
      S     "Bledy_Buffor".Blad_Silnik_Banda_7;
      A     L 0.0;
      AN    "DB_CONNECTOR_BUFF".Banda_17.Silnik_OK;
      S     "Bledy_Buffor".Blad_Silnik_Banda_17;
      A     L 0.0;
      AN    "DB_CONNECTOR_BUFF".Banda_8.Silnik_OK;
      S     "Bledy_Buffor".Blad_Silnik_Banda_8;
      A     L 0.0;
      AN    "DB_CONNECTOR_BUFF".Banda_16.Silnik_OK;
      S     "Bledy_Buffor".Blad_Silnik_Banda_16;
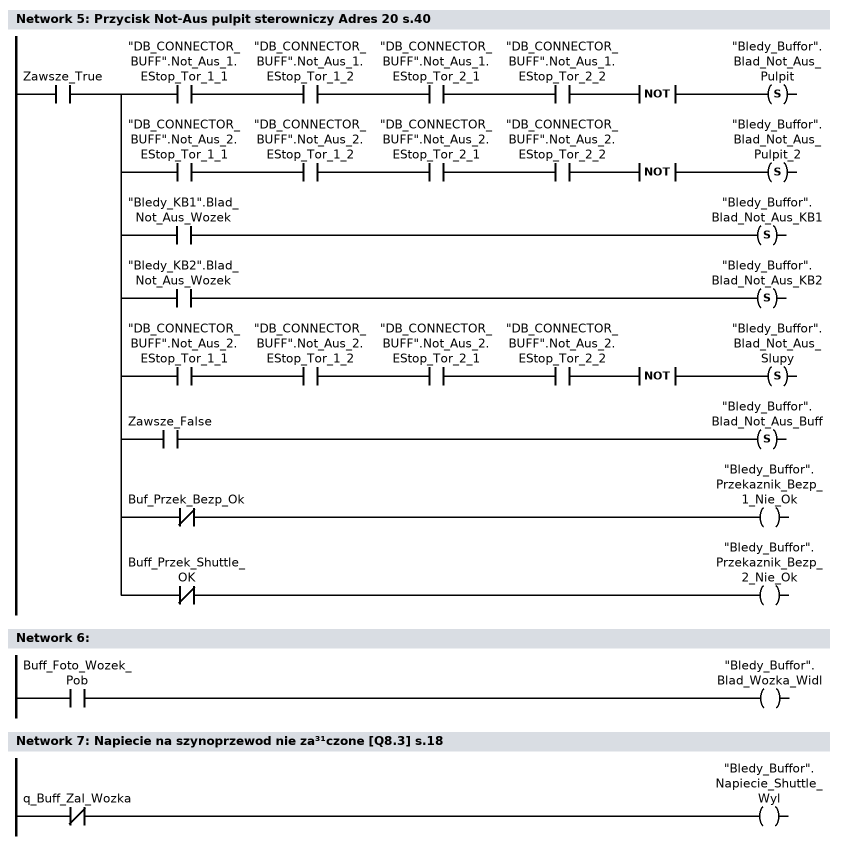
NETWORK
TITLE = Przycisk Not-Aus pulpit sterowniczy Adres 20 s.40
//Bledy not aus
      A     "Zawsze_True";
      =     L 0.0;
      A     L 0.0;
      A     "DB_CONNECTOR_BUFF".Not_Aus_1.EStop_Tor_1_1;
      A     "DB_CONNECTOR_BUFF".Not_Aus_1.EStop_Tor_1_2;
      A     "DB_CONNECTOR_BUFF".Not_Aus_1.EStop_Tor_2_1;
      A     "DB_CONNECTOR_BUFF".Not_Aus_1.EStop_Tor_2_2;
      NOT;
      S     "Bledy_Buffor".Blad_Not_Aus_Pulpit;
      A     L 0.0;
      A     "DB_CONNECTOR_BUFF".Not_Aus_2.EStop_Tor_1_1;
      A     "DB_CONNECTOR_BUFF".Not_Aus_2.EStop_Tor_1_2;
      A     "DB_CONNECTOR_BUFF".Not_Aus_2.EStop_Tor_2_1;
      A     "DB_CONNECTOR_BUFF".Not_Aus_2.EStop_Tor_2_2;
      NOT;
      S     "Bledy_Buffor".Blad_Not_Aus_Pulpit_2;
      A     L 0.0;
      A     "Bledy_KB1".Blad_Not_Aus_Wozek;
      S     "Bledy_Buffor".Blad_Not_Aus_KB1;
      A     L 0.0;
      A     "Bledy_KB2".Blad_Not_Aus_Wozek;
      S     "Bledy_Buffor".Blad_Not_Aus_KB2;
      A     L 0.0;
      A     "DB_CONNECTOR_BUFF".Not_Aus_2.EStop_Tor_1_1;
      A     "DB_CONNECTOR_BUFF".Not_Aus_2.EStop_Tor_1_2;
      A     "DB_CONNECTOR_BUFF".Not_Aus_2.EStop_Tor_2_1;
      A     "DB_CONNECTOR_BUFF".Not_Aus_2.EStop_Tor_2_2;
      NOT;
      S     "Bledy_Buffor".Blad_Not_Aus_Slupy;
      A     L 0.0;
      A     "Zawsze_False";
      S     "Bledy_Buffor".Blad_Not_Aus_Buff;
      A     L 0.0;
      AN    "Buf_Przek_Bezp_Ok";
      =     "Bledy_Buffor".Przekaznik_Bezp_1_Nie_Ok;
      A     L 0.0;
      AN    "Buff_Przek_Shuttle_OK";
      =     "Bledy_Buffor".Przekaznik_Bezp_2_Nie_Ok;
NETWORK
TITLE =
//Blad wozka widlowego
      A     "Buff_Foto_Wozek_Pob";
      =     "Bledy_Buffor".Blad_Wozka_Widl;
NETWORK
TITLE = Napiecie na szynoprzewod nie za³¹czone [Q8.3] s.18
      AN    "q_Buff_Zal_Wozka";
      =     "Bledy_Buffor".Napiecie_Shuttle_Wyl;
END_FUNCTION

FUNCTION "FC_HMI_KB1" : VOID	// FC 121
//Funkcja zawiera elementy wizualizacji i jest skorelowana z blokiem danych 
//db121.
NAME : HMI_KB2
VERSION : 0.1
BEGIN
NETWORK
TITLE =
//Ten Network celowo jest wolny
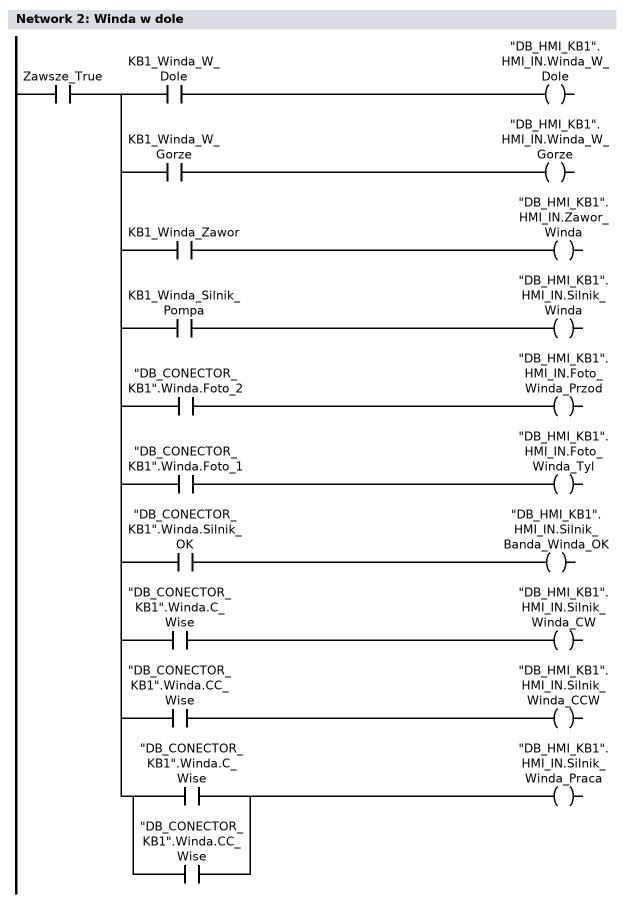
NETWORK
TITLE = Winda w dole
//Wejscia od windy
      A     "Zawsze_True";
      =     L 0.0;
      A     L 0.0;
      A     "KB1_Winda_W_Dole";
      =     "DB_HMI_KB1".HMI_IN.Winda_W_Dole;
      A     L 0.0;
      A     "KB1_Winda_W_Gorze";
      =     "DB_HMI_KB1".HMI_IN.Winda_W_Gorze;
      A     L 0.0;
      A     "KB1_Winda_Zawor";
      =     "DB_HMI_KB1".HMI_IN.Zawor_Winda;
      A     L 0.0;
      A     "KB1_Winda_Silnik_Pompa";
      =     "DB_HMI_KB1".HMI_IN.Silnik_Winda;
      A     L 0.0;
      A     "DB_CONECTOR_KB1".Winda.Foto_2;
      =     "DB_HMI_KB1".HMI_IN.Foto_Winda_Przod;
      A     L 0.0;
      A     "DB_CONECTOR_KB1".Winda.Foto_1;
      =     "DB_HMI_KB1".HMI_IN.Foto_Winda_Tyl;
      A     L 0.0;
      A     "DB_CONECTOR_KB1".Winda.Silnik_OK;
      =     "DB_HMI_KB1".HMI_IN.Silnik_Banda_Winda_OK;
      A     L 0.0;
      A     "DB_CONECTOR_KB1".Winda.C_Wise;
      =     "DB_HMI_KB1".HMI_IN.Silnik_Winda_CW;
      A     L 0.0;
      A     "DB_CONECTOR_KB1".Winda.CC_Wise;
      =     "DB_HMI_KB1".HMI_IN.Silnik_Winda_CCW;
      A     L 0.0;
      A(;
      O     "DB_CONECTOR_KB1".Winda.C_Wise;
      O     "DB_CONECTOR_KB1".Winda.CC_Wise;
      );
      =     "DB_HMI_KB1".HMI_IN.Silnik_Winda_Praca;
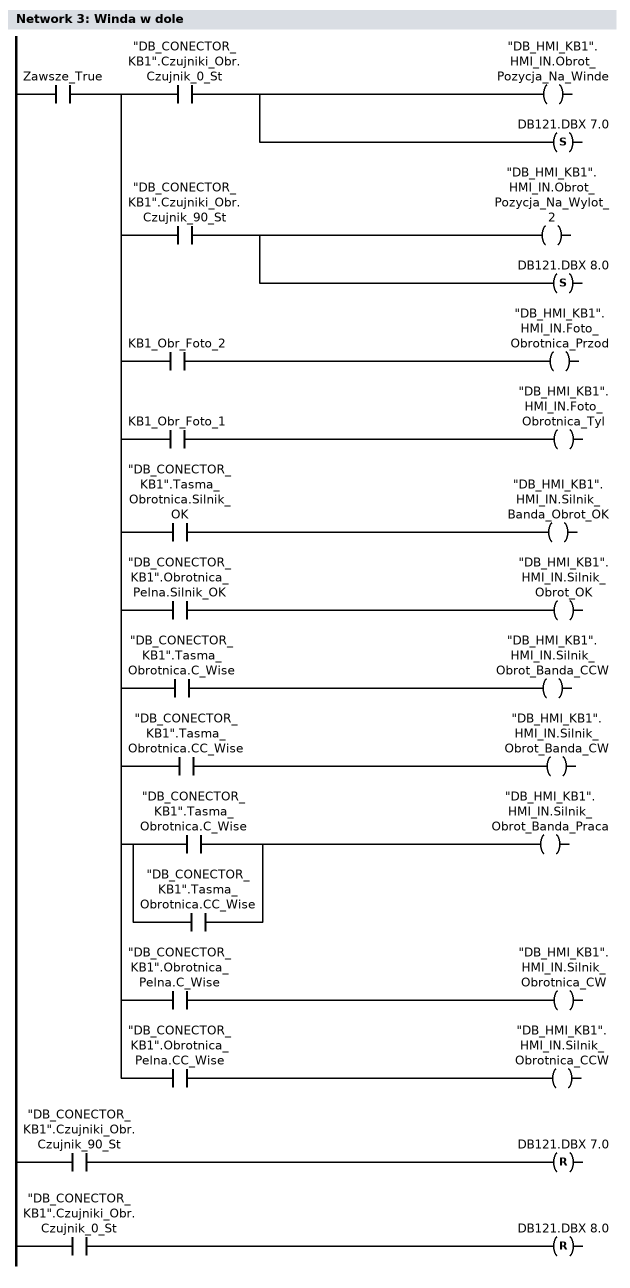
NETWORK
TITLE = Winda w dole
//obrotnica
      A     "Zawsze_True";
      =     L 0.0;
      A     L 0.0;
      A     "DB_CONECTOR_KB1".Czujniki_Obr.Czujnik_0_St;
      =     L 0.1;
      A     L 0.1;
      BLD   102;
      =     "DB_HMI_KB1".HMI_IN.Obrot_Pozycja_Na_Winde;
      A     L 0.1;
      S     DB121.DBX 7.0;
      A     "DB_CONECTOR_KB1".Czujniki_Obr.Czujnik_90_St;
      R     DB121.DBX 7.0;
      NOP   0;
      A     L 0.0;
      A     "DB_CONECTOR_KB1".Czujniki_Obr.Czujnik_90_St;
      =     L 0.1;
      A     L 0.1;
      BLD   102;
      =     "DB_HMI_KB1".HMI_IN.Obrot_Pozycja_Na_Wylot_2;
      A     L 0.1;
      S     DB121.DBX 8.0;
      A     "DB_CONECTOR_KB1".Czujniki_Obr.Czujnik_0_St;
      R     DB121.DBX 8.0;
      NOP   0;
      A     L 0.0;
      A     "KB1_Obr_Foto_2";
      =     "DB_HMI_KB1".HMI_IN.Foto_Obrotnica_Przod;
      A     L 0.0;
      A     "KB1_Obr_Foto_1";
      =     "DB_HMI_KB1".HMI_IN.Foto_Obrotnica_Tyl;
      A     L 0.0;
      A     "DB_CONECTOR_KB1".Tasma_Obrotnica.Silnik_OK;
      =     "DB_HMI_KB1".HMI_IN.Silnik_Banda_Obrot_OK;
      A     L 0.0;
      A     "DB_CONECTOR_KB1".Obrotnica_Pelna.Silnik_OK;
      =     "DB_HMI_KB1".HMI_IN.Silnik_Obrot_OK;
      A     L 0.0;
      A     "DB_CONECTOR_KB1".Tasma_Obrotnica.C_Wise;
      =     "DB_HMI_KB1".HMI_IN.Silnik_Obrot_Banda_CCW;
      A     L 0.0;
      A     "DB_CONECTOR_KB1".Tasma_Obrotnica.CC_Wise;
      =     "DB_HMI_KB1".HMI_IN.Silnik_Obrot_Banda_CW;
      A     L 0.0;
      A(;
      O     "DB_CONECTOR_KB1".Tasma_Obrotnica.C_Wise;
      O     "DB_CONECTOR_KB1".Tasma_Obrotnica.CC_Wise;
      );
      =     "DB_HMI_KB1".HMI_IN.Silnik_Obrot_Banda_Praca;
      A     L 0.0;
      A     "DB_CONECTOR_KB1".Obrotnica_Pelna.C_Wise;
      =     "DB_HMI_KB1".HMI_IN.Silnik_Obrotnica_CW;
      A     L 0.0;
      A     "DB_CONECTOR_KB1".Obrotnica_Pelna.CC_Wise;
      =     "DB_HMI_KB1".HMI_IN.Silnik_Obrotnica_CCW;
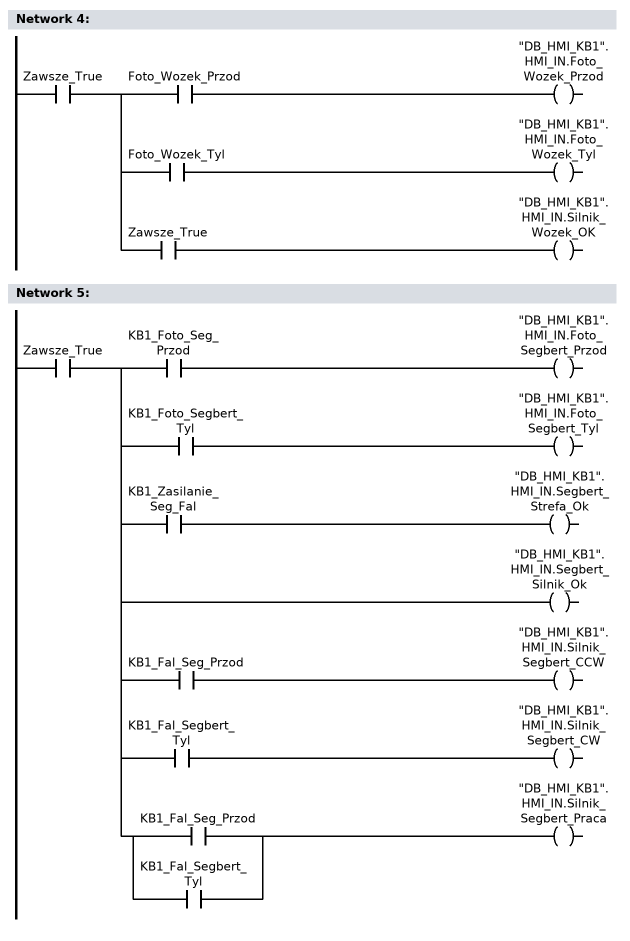
NETWORK
TITLE =
//Wozek
      A     "Zawsze_True";
      =     L 0.0;
      A     L 0.0;
      A     "Foto_Wozek_Przod";
      =     "DB_HMI_KB1".HMI_IN.Foto_Wozek_Przod;
      A     L 0.0;
      A     "Foto_Wozek_Tyl";
      =     "DB_HMI_KB1".HMI_IN.Foto_Wozek_Tyl;
      A     L 0.0;
      A     "Zawsze_True";
      =     "DB_HMI_KB1".HMI_IN.Silnik_Wozek_OK;
NETWORK
TITLE =
//Segbert
//
      A     "Zawsze_True";
      =     L 0.0;
      A     L 0.0;
      A     "KB1_Foto_Seg_Przod";
      =     "DB_HMI_KB1".HMI_IN.Foto_Segbert_Przod;
      A     L 0.0;
      A     "KB1_Foto_Segbert_Tyl";
      =     "DB_HMI_KB1".HMI_IN.Foto_Segbert_Tyl;
      A     L 0.0;
      A     "KB1_Zasilanie_Seg_Fal";
      =     "DB_HMI_KB1".HMI_IN.Segbert_Strefa_Ok;
      A     L 0.0;
      BLD   102;
      =     "DB_HMI_KB1".HMI_IN.Segbert_Silnik_Ok;
      A     L 0.0;
      A     "KB1_Fal_Seg_Przod";
      =     "DB_HMI_KB1".HMI_IN.Silnik_Segbert_CCW;
      A     L 0.0;
      A     "KB1_Fal_Segbert_Tyl";
      =     "DB_HMI_KB1".HMI_IN.Silnik_Segbert_CW;
      A     L 0.0;
      A(;
      O     "KB1_Fal_Seg_Przod";
      O     "KB1_Fal_Segbert_Tyl";
      );
      =     "DB_HMI_KB1".HMI_IN.Silnik_Segbert_Praca;
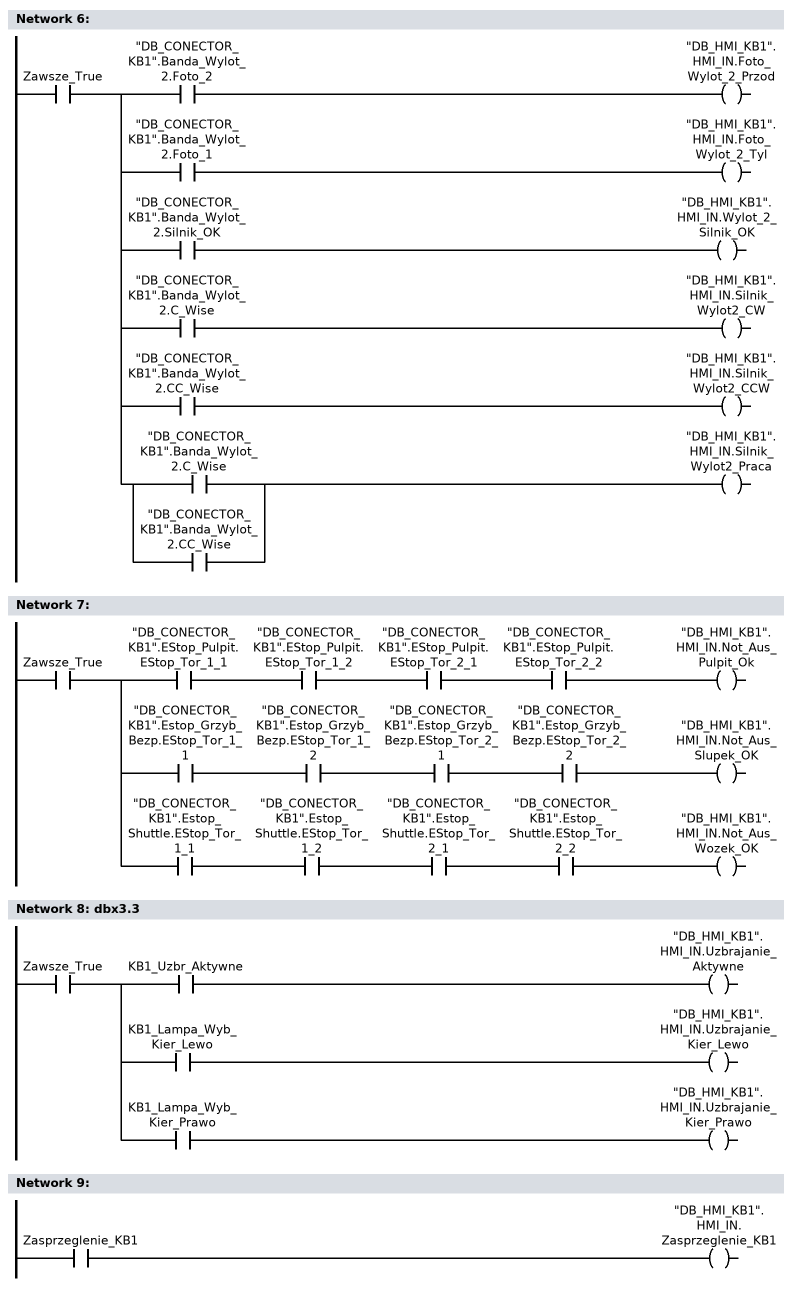
NETWORK
TITLE =
//wylot 2
      A     "Zawsze_True";
      =     L 0.0;
      A     L 0.0;
      A     "DB_CONECTOR_KB1".Banda_Wylot_2.Foto_2;
      =     "DB_HMI_KB1".HMI_IN.Foto_Wylot_2_Przod;
      A     L 0.0;
      A     "DB_CONECTOR_KB1".Banda_Wylot_2.Foto_1;
      =     "DB_HMI_KB1".HMI_IN.Foto_Wylot_2_Tyl;
      A     L 0.0;
      A     "DB_CONECTOR_KB1".Banda_Wylot_2.Silnik_OK;
      =     "DB_HMI_KB1".HMI_IN.Wylot_2_Silnik_OK;
      A     L 0.0;
      A     "DB_CONECTOR_KB1".Banda_Wylot_2.C_Wise;
      =     "DB_HMI_KB1".HMI_IN.Silnik_Wylot2_CW;
      A     L 0.0;
      A     "DB_CONECTOR_KB1".Banda_Wylot_2.CC_Wise;
      =     "DB_HMI_KB1".HMI_IN.Silnik_Wylot2_CCW;
      A     L 0.0;
      A(;
      O     "DB_CONECTOR_KB1".Banda_Wylot_2.C_Wise;
      O     "DB_CONECTOR_KB1".Banda_Wylot_2.CC_Wise;
      );
      =     "DB_HMI_KB1".HMI_IN.Silnik_Wylot2_Praca;
NETWORK
TITLE =
//Not Aus pulpit
//
      A     "Zawsze_True";
      =     L 0.0;
      A     L 0.0;
      A     "DB_CONECTOR_KB1".EStop_Pulpit.EStop_Tor_1_1;
      A     "DB_CONECTOR_KB1".EStop_Pulpit.EStop_Tor_1_2;
      A     "DB_CONECTOR_KB1".EStop_Pulpit.EStop_Tor_2_1;
      A     "DB_CONECTOR_KB1".EStop_Pulpit.EStop_Tor_2_2;
      =     "DB_HMI_KB1".HMI_IN.Not_Aus_Pulpit_Ok;
      A     L 0.0;
      A     "DB_CONECTOR_KB1".Estop_Grzyb_Bezp.EStop_Tor_1_1;
      A     "DB_CONECTOR_KB1".Estop_Grzyb_Bezp.EStop_Tor_1_2;
      A     "DB_CONECTOR_KB1".Estop_Grzyb_Bezp.EStop_Tor_2_1;
      A     "DB_CONECTOR_KB1".Estop_Grzyb_Bezp.EStop_Tor_2_2;
      =     "DB_HMI_KB1".HMI_IN.Not_Aus_Slupek_OK;
      A     L 0.0;
      A     "DB_CONECTOR_KB1".Estop_Shuttle.EStop_Tor_1_1;
      A     "DB_CONECTOR_KB1".Estop_Shuttle.EStop_Tor_1_2;
      A     "DB_CONECTOR_KB1".Estop_Shuttle.EStop_Tor_2_1;
      A     "DB_CONECTOR_KB1".Estop_Shuttle.EStop_Tor_2_2;
      =     "DB_HMI_KB1".HMI_IN.Not_Aus_Wozek_OK;
NETWORK
TITLE = dbx3.3
//Uzbrajanie Aktywne
      A     "Zawsze_True";
      =     L 0.0;
      A     L 0.0;
      A     "KB1_Uzbr_Aktywne";
      =     "DB_HMI_KB1".HMI_IN.Uzbrajanie_Aktywne;
      A     L 0.0;
      A     "KB1_Lampa_Wyb_Kier_Lewo";
      =     "DB_HMI_KB1".HMI_IN.Uzbrajanie_Kier_Lewo;
      A     L 0.0;
      A     "KB1_Lampa_Wyb_Kier_Prawo";
      =     "DB_HMI_KB1".HMI_IN.Uzbrajanie_Kier_Prawo;
NETWORK
TITLE =
//Marka Zasprzeglenia KB1
      A     "Zasprzeglenie_KB1";
      =     "DB_HMI_KB1".HMI_IN.Zasprzeglenie_KB1;
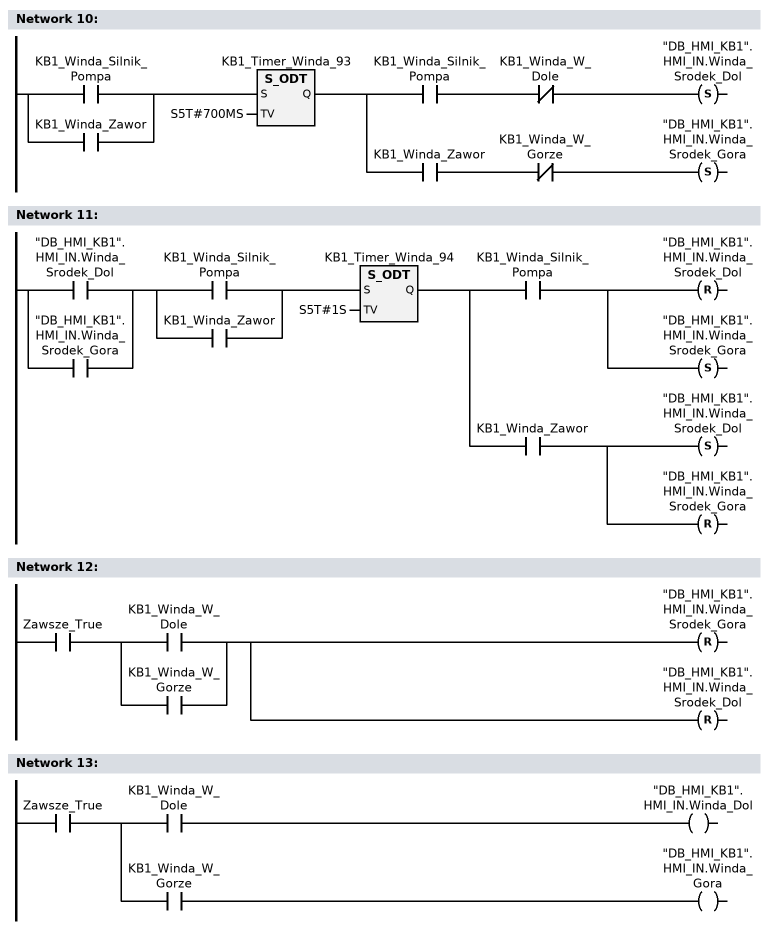
NETWORK
TITLE =
//Animacja windy
      A(;
      O     "KB1_Winda_Silnik_Pompa";
      O     "KB1_Winda_Zawor";
      );
      L     S5T#700MS;
      SD    "KB1_Timer_Winda_93";
      NOP   0;
      NOP   0;
      NOP   0;
      A     "KB1_Timer_Winda_93";
      =     L 0.0;
      A     L 0.0;
      A     "KB1_Winda_Silnik_Pompa";
      AN    "KB1_Winda_W_Dole";
      S     "DB_HMI_KB1".HMI_IN.Winda_Srodek_Dol;
      A     L 0.0;
      A     "KB1_Winda_Zawor";
      AN    "KB1_Winda_W_Gorze";
      S     "DB_HMI_KB1".HMI_IN.Winda_Srodek_Gora;
NETWORK
TITLE =
      A(;
      O     "DB_HMI_KB1".HMI_IN.Winda_Srodek_Dol;
      O     "DB_HMI_KB1".HMI_IN.Winda_Srodek_Gora;
      );
      A(;
      O     "KB1_Winda_Silnik_Pompa";
      O     "KB1_Winda_Zawor";
      );
      L     S5T#1S;
      SD    "KB1_Timer_Winda_94";
      NOP   0;
      NOP   0;
      NOP   0;
      A     "KB1_Timer_Winda_94";
      =     L 0.0;
      A     L 0.0;
      A     "KB1_Winda_Silnik_Pompa";
      R     "DB_HMI_KB1".HMI_IN.Winda_Srodek_Dol;
      S     "DB_HMI_KB1".HMI_IN.Winda_Srodek_Gora;
      A     L 0.0;
      A     "KB1_Winda_Zawor";
      S     "DB_HMI_KB1".HMI_IN.Winda_Srodek_Dol;
      R     "DB_HMI_KB1".HMI_IN.Winda_Srodek_Gora;
NETWORK
TITLE =
//Kasowanie skrajne winda
      A     "Zawsze_True";
      A(;
      O     "KB1_Winda_W_Dole";
      O     "KB1_Winda_W_Gorze";
      );
      R     "DB_HMI_KB1".HMI_IN.Winda_Srodek_Gora;
      R     "DB_HMI_KB1".HMI_IN.Winda_Srodek_Dol;
NETWORK
TITLE =
      A     "Zawsze_True";
      =     L 0.0;
      A     L 0.0;
      A     "KB1_Winda_W_Dole";
      =     "DB_HMI_KB1".HMI_IN.Winda_Dol;
      A     L 0.0;
      A     "KB1_Winda_W_Gorze";
      =     "DB_HMI_KB1".HMI_IN.Winda_Gora;
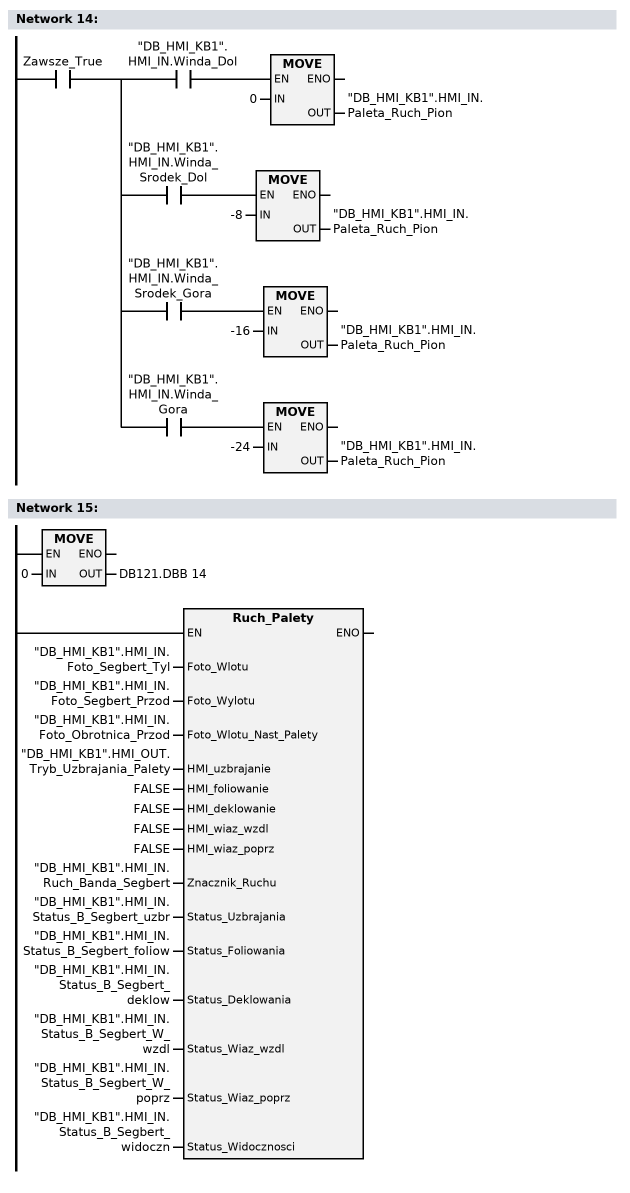
NETWORK
TITLE =
//Ruch windy/palety w pionie
      A     "Zawsze_True";
      =     L 0.0;
      A     L 0.0;
      A     "DB_HMI_KB1".HMI_IN.Winda_Dol;
      JNB   _001;
      L     0;
      T     "DB_HMI_KB1".HMI_IN.Paleta_Ruch_Pion;
_001: NOP   0;
      A     L 0.0;
      A     "DB_HMI_KB1".HMI_IN.Winda_Srodek_Dol;
      JNB   _002;
      L     -8;
      T     "DB_HMI_KB1".HMI_IN.Paleta_Ruch_Pion;
_002: NOP   0;
      A     L 0.0;
      A     "DB_HMI_KB1".HMI_IN.Winda_Srodek_Gora;
      JNB   _003;
      L     -16;
      T     "DB_HMI_KB1".HMI_IN.Paleta_Ruch_Pion;
_003: NOP   0;
      A     L 0.0;
      A     "DB_HMI_KB1".HMI_IN.Winda_Gora;
      JNB   _004;
      L     -24;
      T     "DB_HMI_KB1".HMI_IN.Paleta_Ruch_Pion;
_004: NOP   0;
NETWORK
TITLE =
////Banda Segbert
      L     0;
      T     DB121.DBB 14;
      CALL  "Ruch_Palety" (
           Foto_Wlotu               := "DB_HMI_KB1".HMI_IN.Foto_Segbert_Tyl,
           Foto_Wylotu              := "DB_HMI_KB1".HMI_IN.Foto_Segbert_Przod,
           Foto_Wlotu_Nast_Palety   := "DB_HMI_KB1".HMI_IN.Foto_Obrotnica_Przod,
           HMI_uzbrajanie           := "DB_HMI_KB1".HMI_OUT.Tryb_Uzbrajania_Palety,
           HMI_foliowanie           := FALSE,
           HMI_deklowanie           := FALSE,
           HMI_wiaz_wzdl            := FALSE,
           HMI_wiaz_poprz           := FALSE,
           Znacznik_Ruchu           := "DB_HMI_KB1".HMI_IN.Ruch_Banda_Segbert,
           Status_Uzbrajania        := "DB_HMI_KB1".HMI_IN.Status_B_Segbert_uzbr,
           Status_Foliowania        := "DB_HMI_KB1".HMI_IN.Status_B_Segbert_foliow,
           Status_Deklowania        := "DB_HMI_KB1".HMI_IN.Status_B_Segbert_deklow,
           Status_Wiaz_wzdl         := "DB_HMI_KB1".HMI_IN.Status_B_Segbert_W_wzdl,
           Status_Wiaz_poprz        := "DB_HMI_KB1".HMI_IN.Status_B_Segbert_W_poprz,
           Status_Widocznosci       := "DB_HMI_KB1".HMI_IN.Status_B_Segbert_widoczn);
NETWORK
TITLE =
////Banda Obrotnica 0st
      L     0;
      T     DB121.DBB 15;
      A     DB121.DBX 7.0;
      JCN   et0;
      CALL  "Ruch_Palety" (
           Foto_Wlotu               := "DB_HMI_KB1".HMI_IN.Foto_Obrotnica_Przod,
           Foto_Wylotu              := "DB_HMI_KB1".HMI_IN.Foto_Obrotnica_Tyl,
           Foto_Wlotu_Nast_Palety   := "DB_HMI_KB1".HMI_IN.Foto_Winda_Tyl,
           HMI_uzbrajanie           := "DB_HMI_KB1".HMI_OUT.Tryb_Uzbrajania_Palety,
           HMI_foliowanie           := FALSE,
           HMI_deklowanie           := FALSE,
           HMI_wiaz_wzdl            := FALSE,
           HMI_wiaz_poprz           := FALSE,
           Znacznik_Ruchu           := "DB_HMI_KB1".HMI_IN.Ruch_Banda_Obrotnicy,
           Status_Uzbrajania        := "DB_HMI_KB1".HMI_IN.Status_B_Obr_0st_uzbr,
           Status_Foliowania        := "DB_HMI_KB1".HMI_IN.Status_B_Obr_0st_foliow,
           Status_Deklowania        := "DB_HMI_KB1".HMI_IN.Status_B_Obr_0st_deklow,
           Status_Wiaz_wzdl         := "DB_HMI_KB1".HMI_IN.Status_B_Obr_0st_W_wzdl,
           Status_Wiaz_poprz        := "DB_HMI_KB1".HMI_IN.Status_B_Obr_0st_W_poprz,
           Status_Widocznosci       := "DB_HMI_KB1".HMI_IN.Status_B_Obr_0st_widoczn);
      JU    ok0;
et0:  SET;
      R     "DB_HMI_KB1".HMI_IN.Status_B_Obr_0st_widoczn;
ok0:  NOP   0;
NETWORK
TITLE =
////Banda Obrotnica 90st
      L     0;
      T     DB121.DBB 19;
      A     DB121.DBX 8.0;
      JCN   et90;
      CALL  "Ruch_Palety" (
           Foto_Wlotu               := "DB_HMI_KB1".HMI_IN.Foto_Obrotnica_Przod,
           Foto_Wylotu              := "DB_HMI_KB1".HMI_IN.Foto_Obrotnica_Tyl,
           Foto_Wlotu_Nast_Palety   := "DB_HMI_KB1".HMI_IN.Foto_Wylot_2_Tyl,
           HMI_uzbrajanie           := "DB_HMI_KB1".HMI_OUT.Tryb_Uzbrajania_Palety,
           HMI_foliowanie           := FALSE,
           HMI_deklowanie           := FALSE,
           HMI_wiaz_wzdl            := FALSE,
           HMI_wiaz_poprz           := FALSE,
           Znacznik_Ruchu           := "DB_HMI_KB1".HMI_IN.Ruch_Banda_Obrotnicy,
           Status_Uzbrajania        := "DB_HMI_KB1".HMI_IN.Status_B_Obr_90st_uzbr,
           Status_Foliowania        := "DB_HMI_KB1".HMI_IN.Status_B_Obr_90st_foliow,
           Status_Deklowania        := "DB_HMI_KB1".HMI_IN.Status_B_Obr_90st_deklow,
           Status_Wiaz_wzdl         := "DB_HMI_KB1".HMI_IN.Status_B_Obr_90st_W_wzdl,
           Status_Wiaz_poprz        := "DB_HMI_KB1".HMI_IN.Status_B_Obr_90st_W_popr,
           Status_Widocznosci       := "DB_HMI_KB1".HMI_IN.Status_B_Obr_90st_widocz);
      JU    ok90;
et90: SET;
      R     "DB_HMI_KB1".HMI_IN.Status_B_Obr_90st_widocz;
ok90: NOP   0;
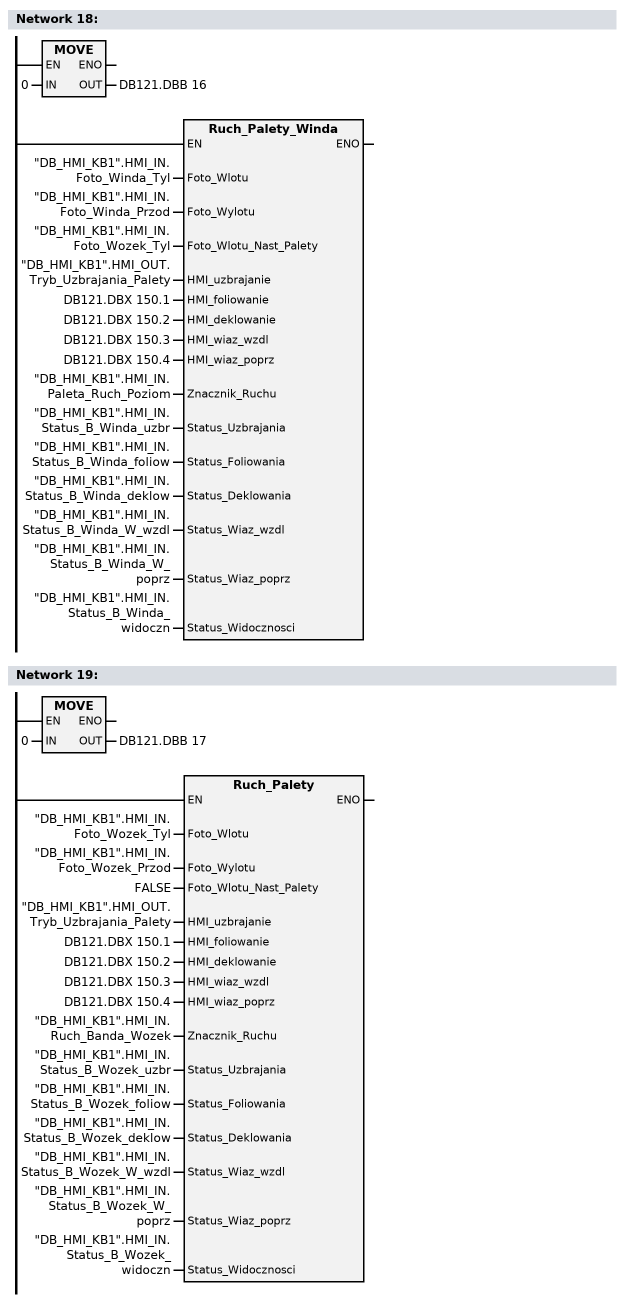
NETWORK
TITLE =
////Banda Winda
      L     0;
      T     DB121.DBB 16;
      CALL  "Ruch_Palety_Winda" (
           Foto_Wlotu               := "DB_HMI_KB1".HMI_IN.Foto_Winda_Tyl,
           Foto_Wylotu              := "DB_HMI_KB1".HMI_IN.Foto_Winda_Przod,
           Foto_Wlotu_Nast_Palety   := "DB_HMI_KB1".HMI_IN.Foto_Wozek_Tyl,
           HMI_uzbrajanie           := "DB_HMI_KB1".HMI_OUT.Tryb_Uzbrajania_Palety,
           HMI_foliowanie           := DB121.DBX 150.1,
           HMI_deklowanie           := DB121.DBX 150.2,
           HMI_wiaz_wzdl            := DB121.DBX 150.3,
           HMI_wiaz_poprz           := DB121.DBX 150.4,
           Znacznik_Ruchu           := "DB_HMI_KB1".HMI_IN.Paleta_Ruch_Poziom,
           Status_Uzbrajania        := "DB_HMI_KB1".HMI_IN.Status_B_Winda_uzbr,
           Status_Foliowania        := "DB_HMI_KB1".HMI_IN.Status_B_Winda_foliow,
           Status_Deklowania        := "DB_HMI_KB1".HMI_IN.Status_B_Winda_deklow,
           Status_Wiaz_wzdl         := "DB_HMI_KB1".HMI_IN.Status_B_Winda_W_wzdl,
           Status_Wiaz_poprz        := "DB_HMI_KB1".HMI_IN.Status_B_Winda_W_poprz,
           Status_Widocznosci       := "DB_HMI_KB1".HMI_IN.Status_B_Winda_widoczn);
NETWORK
TITLE =
////Banda Wozek
      L     0;
      T     DB121.DBB 17;
      CALL  "Ruch_Palety" (
           Foto_Wlotu               := "DB_HMI_KB1".HMI_IN.Foto_Wozek_Tyl,
           Foto_Wylotu              := "DB_HMI_KB1".HMI_IN.Foto_Wozek_Przod,
           Foto_Wlotu_Nast_Palety   := FALSE,
           HMI_uzbrajanie           := "DB_HMI_KB1".HMI_OUT.Tryb_Uzbrajania_Palety,
           HMI_foliowanie           := DB121.DBX 150.1,
           HMI_deklowanie           := DB121.DBX 150.2,
           HMI_wiaz_wzdl            := DB121.DBX 150.3,
           HMI_wiaz_poprz           := DB121.DBX 150.4,
           Znacznik_Ruchu           := "DB_HMI_KB1".HMI_IN.Ruch_Banda_Wozek,
           Status_Uzbrajania        := "DB_HMI_KB1".HMI_IN.Status_B_Wozek_uzbr,
           Status_Foliowania        := "DB_HMI_KB1".HMI_IN.Status_B_Wozek_foliow,
           Status_Deklowania        := "DB_HMI_KB1".HMI_IN.Status_B_Wozek_deklow,
           Status_Wiaz_wzdl         := "DB_HMI_KB1".HMI_IN.Status_B_Wozek_W_wzdl,
           Status_Wiaz_poprz        := "DB_HMI_KB1".HMI_IN.Status_B_Wozek_W_poprz,
           Status_Widocznosci       := "DB_HMI_KB1".HMI_IN.Status_B_Wozek_widoczn);
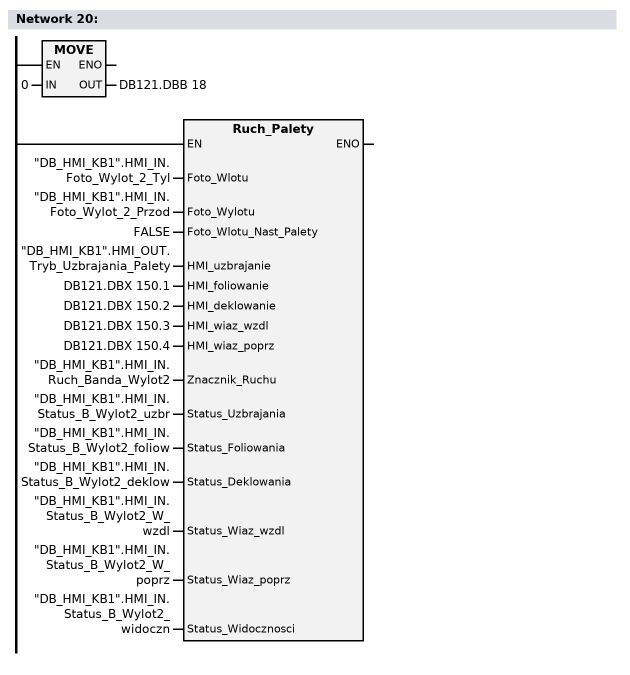
NETWORK
TITLE =
////Banda Wylot2
      L     0;
      T     DB121.DBB 18;
      CALL  "Ruch_Palety" (
           Foto_Wlotu               := "DB_HMI_KB1".HMI_IN.Foto_Wylot_2_Tyl,
           Foto_Wylotu              := "DB_HMI_KB1".HMI_IN.Foto_Wylot_2_Przod,
           Foto_Wlotu_Nast_Palety   := FALSE,
           HMI_uzbrajanie           := "DB_HMI_KB1".HMI_OUT.Tryb_Uzbrajania_Palety,
           HMI_foliowanie           := DB121.DBX 150.1,
           HMI_deklowanie           := DB121.DBX 150.2,
           HMI_wiaz_wzdl            := DB121.DBX 150.3,
           HMI_wiaz_poprz           := DB121.DBX 150.4,
           Znacznik_Ruchu           := "DB_HMI_KB1".HMI_IN.Ruch_Banda_Wylot2,
           Status_Uzbrajania        := "DB_HMI_KB1".HMI_IN.Status_B_Wylot2_uzbr,
           Status_Foliowania        := "DB_HMI_KB1".HMI_IN.Status_B_Wylot2_foliow,
           Status_Deklowania        := "DB_HMI_KB1".HMI_IN.Status_B_Wylot2_deklow,
           Status_Wiaz_wzdl         := "DB_HMI_KB1".HMI_IN.Status_B_Wylot2_W_wzdl,
           Status_Wiaz_poprz        := "DB_HMI_KB1".HMI_IN.Status_B_Wylot2_W_poprz,
           Status_Widocznosci       := "DB_HMI_KB1".HMI_IN.Status_B_Wylot2_widoczn);
END_FUNCTION

FUNCTION "FC_HMI_KB2" : VOID	// FC 122
//Funkcja zawiera elementy wizualizacji i jest skorelowana z blokiem danych 
//db122.
NAME : HMI_KB2
VERSION : 0.1
BEGIN
NETWORK
TITLE =
//Ten Network celowo jest wolny
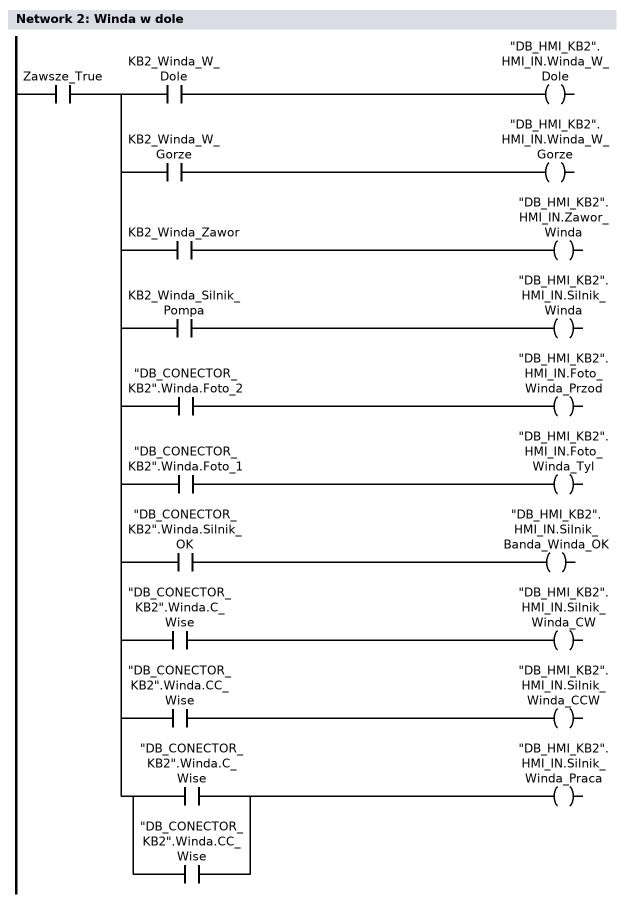
NETWORK
TITLE = Winda w dole
//Wejscia od windy
      A     "Zawsze_True";
      =     L 0.0;
      A     L 0.0;
      A     "KB2_Winda_W_Dole";
      =     "DB_HMI_KB2".HMI_IN.Winda_W_Dole;
      A     L 0.0;
      A     "KB2_Winda_W_Gorze";
      =     "DB_HMI_KB2".HMI_IN.Winda_W_Gorze;
      A     L 0.0;
      A     "KB2_Winda_Zawor";
      =     "DB_HMI_KB2".HMI_IN.Zawor_Winda;
      A     L 0.0;
      A     "KB2_Winda_Silnik_Pompa";
      =     "DB_HMI_KB2".HMI_IN.Silnik_Winda;
      A     L 0.0;
      A     "DB_CONECTOR_KB2".Winda.Foto_2;
      =     "DB_HMI_KB2".HMI_IN.Foto_Winda_Przod;
      A     L 0.0;
      A     "DB_CONECTOR_KB2".Winda.Foto_1;
      =     "DB_HMI_KB2".HMI_IN.Foto_Winda_Tyl;
      A     L 0.0;
      A     "DB_CONECTOR_KB2".Winda.Silnik_OK;
      =     "DB_HMI_KB2".HMI_IN.Silnik_Banda_Winda_OK;
      A     L 0.0;
      A     "DB_CONECTOR_KB2".Winda.C_Wise;
      =     "DB_HMI_KB2".HMI_IN.Silnik_Winda_CW;
      A     L 0.0;
      A     "DB_CONECTOR_KB2".Winda.CC_Wise;
      =     "DB_HMI_KB2".HMI_IN.Silnik_Winda_CCW;
      A     L 0.0;
      A(;
      O     "DB_CONECTOR_KB2".Winda.C_Wise;
      O     "DB_CONECTOR_KB2".Winda.CC_Wise;
      );
      =     "DB_HMI_KB2".HMI_IN.Silnik_Winda_Praca;
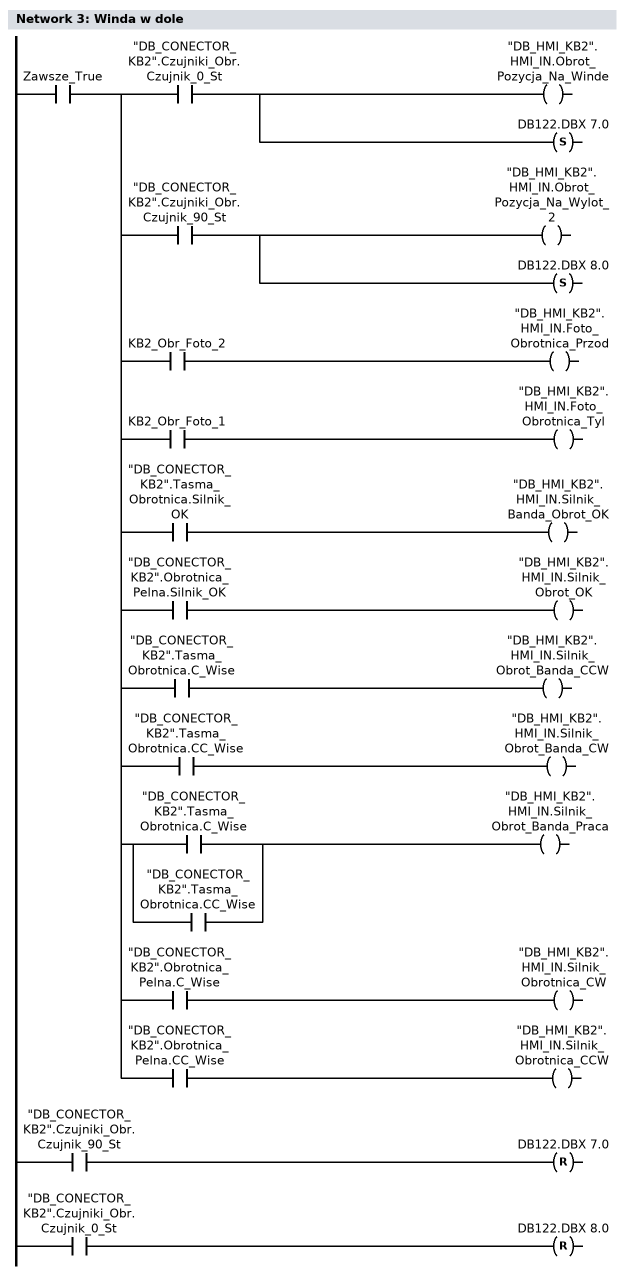
NETWORK
TITLE = Winda w dole
//obrotnica
      A     "Zawsze_True";
      =     L 0.0;
      A     L 0.0;
      A     "DB_CONECTOR_KB2".Czujniki_Obr.Czujnik_0_St;
      =     L 0.1;
      A     L 0.1;
      BLD   102;
      =     "DB_HMI_KB2".HMI_IN.Obrot_Pozycja_Na_Winde;
      A     L 0.1;
      S     DB122.DBX 7.0;
      A     "DB_CONECTOR_KB2".Czujniki_Obr.Czujnik_90_St;
      R     DB122.DBX 7.0;
      NOP   0;
      A     L 0.0;
      A     "DB_CONECTOR_KB2".Czujniki_Obr.Czujnik_90_St;
      =     L 0.1;
      A     L 0.1;
      BLD   102;
      =     "DB_HMI_KB2".HMI_IN.Obrot_Pozycja_Na_Wylot_2;
      A     L 0.1;
      S     DB122.DBX 8.0;
      A     "DB_CONECTOR_KB2".Czujniki_Obr.Czujnik_0_St;
      R     DB122.DBX 8.0;
      NOP   0;
      A     L 0.0;
      A     "KB2_Obr_Foto_2";
      =     "DB_HMI_KB2".HMI_IN.Foto_Obrotnica_Przod;
      A     L 0.0;
      A     "KB2_Obr_Foto_1";
      =     "DB_HMI_KB2".HMI_IN.Foto_Obrotnica_Tyl;
      A     L 0.0;
      A     "DB_CONECTOR_KB2".Tasma_Obrotnica.Silnik_OK;
      =     "DB_HMI_KB2".HMI_IN.Silnik_Banda_Obrot_OK;
      A     L 0.0;
      A     "DB_CONECTOR_KB2".Obrotnica_Pelna.Silnik_OK;
      =     "DB_HMI_KB2".HMI_IN.Silnik_Obrot_OK;
      A     L 0.0;
      A     "DB_CONECTOR_KB2".Tasma_Obrotnica.C_Wise;
      =     "DB_HMI_KB2".HMI_IN.Silnik_Obrot_Banda_CCW;
      A     L 0.0;
      A     "DB_CONECTOR_KB2".Tasma_Obrotnica.CC_Wise;
      =     "DB_HMI_KB2".HMI_IN.Silnik_Obrot_Banda_CW;
      A     L 0.0;
      A(;
      O     "DB_CONECTOR_KB2".Tasma_Obrotnica.C_Wise;
      O     "DB_CONECTOR_KB2".Tasma_Obrotnica.CC_Wise;
      );
      =     "DB_HMI_KB2".HMI_IN.Silnik_Obrot_Banda_Praca;
      A     L 0.0;
      A     "DB_CONECTOR_KB2".Obrotnica_Pelna.C_Wise;
      =     "DB_HMI_KB2".HMI_IN.Silnik_Obrotnica_CW;
      A     L 0.0;
      A     "DB_CONECTOR_KB2".Obrotnica_Pelna.CC_Wise;
      =     "DB_HMI_KB2".HMI_IN.Silnik_Obrotnica_CCW;
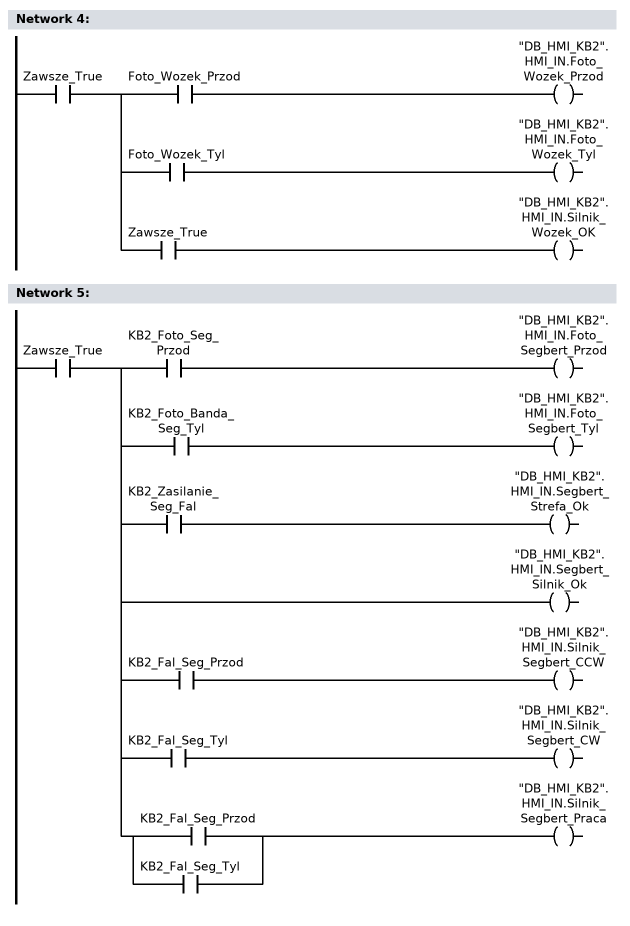
NETWORK
TITLE =
//Wozek
      A     "Zawsze_True";
      =     L 0.0;
      A     L 0.0;
      A     "Foto_Wozek_Przod";
      =     "DB_HMI_KB2".HMI_IN.Foto_Wozek_Przod;
      A     L 0.0;
      A     "Foto_Wozek_Tyl";
      =     "DB_HMI_KB2".HMI_IN.Foto_Wozek_Tyl;
      A     L 0.0;
      A     "Zawsze_True";
      =     "DB_HMI_KB2".HMI_IN.Silnik_Wozek_OK;
NETWORK
TITLE =
//Segbert
//
      A     "Zawsze_True";
      =     L 0.0;
      A     L 0.0;
      A     "KB2_Foto_Seg_Przod";
      =     "DB_HMI_KB2".HMI_IN.Foto_Segbert_Przod;
      A     L 0.0;
      A     "KB2_Foto_Banda_Seg_Tyl";
      =     "DB_HMI_KB2".HMI_IN.Foto_Segbert_Tyl;
      A     L 0.0;
      A     "KB2_Zasilanie_Seg_Fal";
      =     "DB_HMI_KB2".HMI_IN.Segbert_Strefa_Ok;
      A     L 0.0;
      BLD   102;
      =     "DB_HMI_KB2".HMI_IN.Segbert_Silnik_Ok;
      A     L 0.0;
      A     "KB2_Fal_Seg_Przod";
      =     "DB_HMI_KB2".HMI_IN.Silnik_Segbert_CCW;
      A     L 0.0;
      A     "KB2_Fal_Seg_Tyl";
      =     "DB_HMI_KB2".HMI_IN.Silnik_Segbert_CW;
      A     L 0.0;
      A(;
      O     "KB2_Fal_Seg_Przod";
      O     "KB2_Fal_Seg_Tyl";
      );
      =     "DB_HMI_KB2".HMI_IN.Silnik_Segbert_Praca;
